(* CODESYS project Brau-Codesys
   Author: Robert Budgen
   Company: Burkert-Canada
   CompiledLibraryCompatibilityVersion: e!COCKPIT
   DefaultNamespace: Brau
   LanguageModelAttribute: qualified-access-only
   Placeholder: Brau
   Title: Brau
   Version: 3.0.0.49

Project tree, tasks and I/O mapping:
  libraries: CAA Types Extern, 3.5.17.0 (CAA Technical Workgroup); CAA Behaviour Model, 3.5.19.0 (CAA Technical Workgroup); CAA FB Factory, 3.5.19.0 (CAA Technical Workgroup); Standard, 3.5.18.0 (System); Util, 3.5.21.0 (System); CmpBitmapPool, 3.5.17.0 (System); VisuDialogs, * (System); MemoryUtils, 3.5.18.0 (3S - Smart Software Solutions GmbH); CAA Memory, 3.5.17.0 (CAA Technical Workgroup); SysTimeRtc, 3.5.20.0 (System); CAA CiA 405, 4.1.0.0 (CAA Technical Workgroup); IoDrvEtherNetIPAdapter, 4.8.0.0 (CODESYS); IoDrvEtherNetIP, 4.8.0.0 (CODESYS); BUILDING, 1.0.0.0 (OSCAT); BASIC, 3.3.4.0 (OSCAT); FloatingPointUtils, 4.0.0.0 (System); 3S CANopenStack, 4.3.0.0 (CODESYS); IoDrvModbusTCP, 4.5.0.0 (CODESYS); Recipe Management, * (System); Burkert Device Library, 1.0.0.102 (Burkert)
  25 Interfaces/
    interface IcSensorProvider: GetSensorRef
  50 Functions/
    Burkert Library/
      function Alarm_Window_Convert [ST]
      function ASi_8694_Mapping [CFC]
      function block b8619_CND_FB [ST]
      function block B8619_Input_FB [ST]
      function block B8619_Main_FB [ST]
      function block b8619_PH_ORP_FB [ST]
      function Build_ORF_Index [ST]
      function FlowWave_Mapping [LD]
      function Tempered_Look_UP [ST]
    function DaySeconds [?]
  90 Task Enums/
    data type eCLT_Task
    data type eGR_Task
    data type eHLT_Task
    data type eKT_Task
    data type eLT_Task
    data type eMM_Task
    data type eWP_Task
    Level_3/
  95 Base Mappings/
    Level_0/
      data type IoLink_Mapping
      data type ME44AI_Mapping
      data type ME44AO_Mapping
      data type ME44DI_Mapping
      data type ME44DO_Mapping
      data type me64_Mapping
    Level_1/
      data type ACV_Mapping_1
      data type AIT_Mapping_1
      data type b8653_mapping
      data type BCV_Mapping_1
      data type cSensor_Mapping
      data type dACV_Mapping
      data type dBCV_Mapping
      data type DI_Mapping
      data type Do_Mapping
      data type FIT_Mapping_1
      data type LS_Mapping_1
      data type PT_Mapping_1
      data type s8050_Mapping
      data type s8228_Mapping
      data type s8312_Mapping
      data type s8412_Mapping
      data type SV_Mapping
      data type TT_Mapping_1
      data type v336x_Mapping
    Level_2/
      data type Analog_Pump_Mapping
      data type mPump_Mapping
      data type PID_Mapping_1
      data type Stack_Light_Mapping
      data type VFD_Mapping
    Level_3/
      data type Alarm_Offset_Mapping
      data type Brite_Mapping_1
      data type Fermenter_Mapping_1
  AL1342
  CanOpen_8694
  Level_3/
    Fermenter
  function block ACV_Temp_Loop_UDFB [CFC]
  function block AODD_UDFB [CFC]
  Asi/
    function block AC2916_AIT [LD]
    function block ACV_ASI_CTRL_UDFB [?]
    function block B8681_ASI_UDFB [CFC]
    function block BCV_ASI_CTRL_UDFB [?]
  function block Basic_Temp_LOOP [CFC]
  function block BCV_Temp_Loop_UDFB [CFC]
  Burkert Library/
    Burkert/
      function eDip_ME44_AO [ST]
      function eDip_ME44_DO_Analog [ST]
      function eDip_ME44_DO [ST]
      function block eDip_ReadSingleItem [ST]
      function block ME43_SDO [ST]: Direct_Write
      function ME44_DI [ST]
    CanOpen/
    eDip/
      function block eDip_8605_CTRL [ST]: Parse_TX
      function eDip_ME44_AI [ST]
      function eDip_ME44_DI [ST]
    function block Parse_DDO [ST]
    function block Parse_DSO [ST]
  function block Chase_Master_Rate_UDFB [SFC]
  function block Chase_Master_UDFB [SFC]
  function block Chase_Slave_UDFB [ST]
  Level_0_Remote_IO/
    function block AL1340_UDFB [ST]
    function block AL1342_UDFB [ST]
    MicroControl/
      function MC4AI [ST]
  Level_1_Devices/
    function block Analog_Control_UDFB [LD]
    Burkert Library/
      function block Analog_Alarm_UDFB [ST]: run
      function block Analog_Sensor_UDFB [?]
      function block B8619_UDFB [CFC]: PH
      function block Basic_ACV_UDFB [?]
      function block Basic_BCV_UDFB [ST]: Eval_Output, Eval_Ready, Eval_Status
      function block Basic_FIT [?]
      function block BCV_CTRL_UDFB [?]
      CanOpen/
        function block CanOpen_8098 [CFC]
        function block CanOpen_8228 [ST]
        function block CanOpen_8691 [?]
        function block CanOpen_8694 [?]
        function block CanOpen_MS02 [ST]
        function block CanOpen_MS03 [ST]
        function block CanOpen_MS04 [ST]
        function block CanOpen_MS05 [ST]
      eDip/
        function block eDip_336x [ST]
        function block eDip_8098_CTRL [ST]
        function block eDip_8228_MEx3 [ST]
        function block eDip_8312 [ST]
        function block eDip_8412 [ST]
        function block eDip_8681_UDFB [CFC]
        function block eDIP_SDO_Manager [CFC]
      function block FIT_Count_UDFB [?]
      function block FIT_Rate_UDFB [?]
      function block FIT_UDFB [?]
      IoLink/
        function block s8050_UDFB [CFC]
      function block LS_UDFB [ST]
      function SV_Fun [CFC]
    function block Stack_Lights_4Way [CFC]
  Level_2_Controls/
    function block Analog_Batch_Pump [CFC]: Set_Status
    function block Batch [ST]: AUX
    function block Condensate_Trap_UDFB [CFC]: Positions, Purge, Status
    function block DofMaster [ST]
    function block Duplex_VFD [ST]: Outputs
    function block PID_UDFB [CFC]
    function block Quick_Mix_UDFB [SFC]: Auto_active, Aux_active, End_active, FIT_Reset_active, Init_active, Init_entry, Main_Rate_active, OFF_active, OFF_entry, Paused_active, Ramp_Down_active, Ramp_Up_active, Start_active, Start_entry, System_Test_active, System_Text_entry
    function block Rate_Batch [ST]
    function block SW_CTRL_ACV [ST]
    function block SW_CTRL [ST]
    function block Tempered_Line_4_Valve [ST]: Alarms, AUX, Math, PID_CTRL, Task_Calibrate, Task_Prime, Task_Run
  Level_3/
  program PLC_TIME [ST]
  Simulators/
    function block c8691_CanOpen_Sim [ST]
    function c8694_CanOpen_Sim [ST]
    function CanOpen_8694_Data_Sim [ST]
    function block Contactor_Sim [ST]
    function Edip_8691_Sim [ST]
    function Edip_8694_Data_Sim [ST]
    function eDip_ME44_DI_Count_Sim [ST]
    function eDip_ME44_DI_Hz_Sim [ST]
    function FIT_Sim [ST]
    function Mix_Sim [ST]
    function TT_SIM [ST]
    function block Vacon_VFD_SIM [ST]
  function block Tempered_Mix_eDip_UDFB [CFC]
  function block Tempered_Mix_UDFB [CFC]
  function block Transfer_ACV_FIT_UDFB [CFC]
  function block Transfer_ACV_VFD_FIT_UDFB [CFC]
  function block Transfer_BCV_FIT_UDFB [CFC]
  function block Transfer_BCV_VFD_FIT_UDFB [CFC]
  Vessels/
  In Burkert Device Library/
    Base_Declarations/
      data type cBase_FIT
      Level_1/
    Level_0_Remote_IO/
    LeveL_1/
      data type cACV
      data type cAIT
      data type cAnalog_Sensor
      data type cBCV
      data type cFIT
      IO-Link/
        data type c8050
      Networked/
      data type SV_DUT
    To be Sorted/
      data type ACV_eDip
      data type Alarm_Config
      data type Alarm_Window
      data type Analog_scale
      data type AODD_DUT
      data type Asi_Node_DUT
      data type b8619_CND_DUT
      data type b8619_Inputs_DUT
      data type b8619_Main_DUT
      data type b8619_PH_DUT
      data type B8691_Asi_DUT
      data type c8694_PDin
      data type cFLOWave_DUT
      data type CND_8619
      data type cSDO_DUT
      data type eDip_8681_DUT
      data type eDip_DDO
      data type eDip_DSO
      data type eDip_MFC_DUT
      data type FV_DUT
      data type HLT_Blending_DUT
      data type HLT_Chase_DUT
      data type PH_8619
      data type PT_Config_DUT
      data type SDO
      data type Steam_Set_Config_DUT
      data type Steam_Set_DUT
      data type TT_Config_DUT
      data type Vessel_Config_Dut
      data type Word_as_Real_DUT
  Level_0/
    Adam_6050/
      data type cAdam_6050_MBTCP
    Adam_6052/
      data type cAdam_6052_Control
      data type cAdam_6052_MBTCP
    Adam_6217/
    Adam_6250/
    IO-Link/
      data type c8694_Io_Link
      data type cIFM_AL1340
      data type cIFM_AL1342
    data type MicroControl_4AI
    SIO-MB04RTDS/
      data type cMB0_RTD
    SIO-MB12CDR/
      data type cSIO_MB12CDR
  Level_1_Devices/
    data type cContactor
    data type DI_DUT
  Level_2_Functions/
    data type Analog_Control_DUT
    data type cAnalog_Batch_Pump
    data type cCondensate_Trap
    data type cDuplex
    data type cFilters
    data type cStack_Light
  Level_3/
    Brewery/
      data type Brewery_Config_DUT
    data type cBatch
    data type cDOF_Master
  Burkert Library/
    data type IFM_Status
    data type ORF
    data type uACV_Mode
    data type uACV_Status
    data type uAIT_Mode
    data type uBCV_Mode
    data type uNamur
    data type uNord_Data_In
    data type uNord_Status_Word
    data type uSensor_Status
  data type Bytes_2_Int
  data type bytes_2_real
  data type Bytes_DWord
  data type Bytes_Word
  data type eKT_Mode
  Level_1/
    data type uAnalog_Pump_Modes
    data type uAnalog_Pump_Status
    data type uContactor_Modes
    data type uDI_Mode
    data type uDI_Status
    data type uDo_Modes
    data type uHOA_Mode
    data type uM_Pump_Modes
    data type uM_Pump_Status
    data type uVFD_Mode
    data type uVFD_Status
  data type REAL_2_WORD
  data type uBatch_Status
  data type uBatch_Task
  data type uBatch_Transfer_Mode
  data type uBrite_Modes
  data type uBrite_Status
  data type uBrite_Status
  data type uChase_Status
  data type uCLT_Mode
  data type uCLT_Status
  data type uCLT_Task
  data type uContactor_Status
  data type uFermenter_Modes
  data type uFermenter_Status
  data type uFilter_Manager_Modes
  data type uFilterMode
  data type uGR_Status
  data type uGR_Task
  data type uHighSpeed_Tempered_Mode
  data type uHighSpeed_Tempered_Status
  data type uHighSpeed_Tempered_Task
  data type uHLT_Mode
  data type uHLT_Status
  data type uHLT_Task
  data type uKT_Mode
  data type uKT_Status
  data type uKT_Task
  data type uLT_Mode
  data type uLT_Status
  data type uLT_Task
  data type uMM_Mode
  data type uMM_Task
  data type uPID_Modes
  data type uPID_Status
  data type uQuick_Mix_Modes
  data type uService_Water_Destination
  data type uTempered_Modes
  data type uTempered_Status
  data type uTempered_Tasks
  data type uUser_Confirm
  data type uWP_Mode
  data type uWP_Modes
  data type uWP_Status
  data type uWP_Task
  data type WORD_2_Real
  data type AIT_Transfer_Modes
  Burkert Library/
    Brewery/
    data type e_8681_Modes
    data type eAODD_Modes
    data type eB336x_Modes
    data type eConfig_startTune
    data type eHOA_Modes
    Level_1/
      data type ACV_Modes
      data type AIT_Modes
      data type eBCV_Modes
      data type TT_Modes
    data type LS_Modes
    data type Positioner_Modes
    data type PT_Modes
    data type Reset_Relay_Mode
  data type CLT_Modes
  data type Command_Modes
  data type eChase_Mode
  data type Fan_Modes
  data type FIT_Transfer_Modes
  data type FIT_VFD_Transfer_Modes
  Level_0/
  Level_1/
    data type eVFD_Modes
  Level_3/
    data type eBrite_Modes
    data type eCLT_Modes
    data type eFermenter_Modes
    data type eGR_Modes
    data type eHLT_Modes
    data type eKT_Modes
    data type eLT_Modes
    data type eMM_Modes
    data type eRCP_Mode
    data type eWP_Modes
    data type FV_Modes
    data type HLT_Blending_Modes
    data type KTWP_Modes
  data type Steam_Condensate_Modes
  data type Steam_Modes
  data type Temp_loop_Modes
  Burkert Library/
    Level_1/
      data type eACV_Status
      data type eBCV_Status
      data type eSensor_Status
  data type e8691_ValveMode
  data type e8691_xTuneStatus
  data type e8694_xTuneStatus
  data type eB8681_Status
  data type eCurrentOpMode
  data type eNamur107
  data type eORF_Status
  Level_1/
    data type Contactor_Status
    data type DI_Status
    data type DO_Status
    data type eAnalog_Pump_Status
    data type eAODD_Status
    data type eM_Pump_Status
    data type eVFD_Status
    data type VFD_Fault_Status
  Level_2/
    data type eCondensate_Status
    data type eFilter_Manager_Status
    data type eFilter_Status
  Level_3/
  data type SDO_Error_Codes
  Vessels/
    data type eBrite_Status
    data type eCLT_Status
    data type eHLT_Status
    data type eKT_Status
    data type eLT_Status
    data type eMM_Status
    data type eWP_Status
  data type eHLT_Notifications
  data type eMM_Notifications
  function GetLibVersion [ST]
  function GetLibVersionNumber [ST]
  function IsLibReleased [ST]
  function GetBooleanProperty [ST]
  function GetCompany [ST]
  function GetTextProperty2 [ST]
  function GetTextProperty [ST]
  function GetTitle [ST]
  function GetVersion [ST]
  function GetVersionProperty [ST]
  function block FB_PositionTracker [ST]
  function fbMidPoint [ST]
  function RCP_Manager [ST]
  function block Virtual_FIT [CFC]
  Burkert Library/
    ASi/
      function block ASi_8694_HMI_Sync_UDFB [?]
    Level_0/
    Level_1/
      function block ACV_HMI_Sync_UDFB [?]
      function block AIT_HMI_Sync_UDFB [?]
      function block B8050_HMI_Sync_UDFB [?]
      function block BCV_HMI_Sync_UDFB [?]
      function block c8691_HMI_Sync_UDFB [?]
      function block c8694_HMI_Sync_UDFB [?]
      function block DI_HMI_Sync_UDFB [?]
      function block FIT_HMI_Sync_UDFB [?]
      function block GS20_VFD_HMI_Sync [?]
      function block s336x_HMI_Sync [?]
      function block s8050_HMI_Sync [?]
      function block s8098_HMI_Sync_UDFB [?]
      function block s8312_HMI_Sync [?]
      function block SV_HMI_Sync [?]
      function block Vacon_HMI_Sync_UDFB [?]
  Level_1/
    function block Analog_Pump_HMI_Sync [?]
    function block Contactor_HMI_Sync_UDFB [?]
    function block Eaton_VFD_HMI_Sync [?]
    function block M_Pump_HMI_Sync [?]
  Level_2/
    function block PID_HMI_Sync_UDFB [?]
  Level_3/
    function block Brite_HMI_Sync [?]
    function block Fermenter_HMI_Sync [?]
  data type ASi_8694
  data type ASi_8694_PDO
  Burkert Librarry/
    Level_0/
    Level_1/
      data type HMI_8050
      data type HMI_AIT
      data type HMI_BCV
      data type HMI_FIT
      data type HMI_VFD_GS20_DUT
      data type HMI_VFD_Vacon_DUT
  Level_1/
    data type HMI_Analog_Pump
    data type HMI_Contactor_DUT
    data type HMI_M_Pump
    data type HMI_VFD_Eaton_DUT
  Level_2/
    data type HMI_PID
  Level_3/
    data type HMI_Brite
    data type HMI_Fermenter
  function block AC2916 [CFC]
  function block Asi_GW_FUN [ST]
  function f_Fermenter_To_NVL [ST]
  data type eAnalog_Control_Modes
  data type eFilter_Manager_Modes
  data type eFilter_Mode
  data type eTempered_Modes
  function Adam_6050_FB [LD]
  function Adam_6250 [ST]
  function block MB0_RTD [ST]
  function block SIO_MB12CDR [ST]
  function block Contactor [ST]: Status
  function block Contactor_Control_UDFB [CFC]: Status
  function block DI_UDFB [CFC]
  function block DO_UDFB [CFC]
  function block Analog_Pump [ST]: Status
  function block Eaton_DM1 [ST]: Control, Data_IN, Data_Out, Status
  function block Nord_VFD_UDFB [CFC]
  function block Vacon_100 [ST]: Control, Data_IN, Data_Out, Data_Sim, Status
  function block VFD_GS20_UDFB [?]: Status
  function block VFD_GS2_UDFB [LD]
  function block VFD_Vacon100_UDFB [?]
  function block Wago_750_455 [LD]
  function block Wago_750_NAMUR_NE43 [?]
  data type VFD_CONTROL
  data type VFD_GS2_DUT
  data type VFD_WEG_DUT
  data type cFilter
  data type cFilter_Manager
  data type Quick_Mix_Control
  data type cPID_DUT
  data type cTempered_Line_Data
  function block Brite_1_UDFB [CFC]
  function block Brite_2_UDFB [CFC]
  function block Brite_3_UDFB [CFC]
  function block Fermenter_1_UDFB [CFC]
  function block Fermenter_2_UDFB [CFC]
  function block Fermenter_3_UDFB [CFC]
  program CLT [ST]
  KT/
  LT/
  MM/
  WP/
  program Grain_Room_Hopper_1Conveyor [ST]
  Controls/
  program HLT_2Pump_2Mix [ST]
  program HLT_2Pump_2Mix_OLD [CFC]
  function block HLT_PID_Manager [CFC]
  function block HLT_Status_Manager [?]
  function block HLT_Task_Manager [CFC]
  function block HLT_Tasks_OLD [SFC]
  function block HLT_Valve_Manager [CFC]
  function block HLT_VFD_Ctrl [CFC]
  function block Service_Water [SFC]
  function block Service_Water_Manager [CFC]
  Tasks/
  data type ceDip_ME44_DI
  data type cME44_DO
  data type cME44_DO_TX
  data type cVFD_Eaton_DUT
  data type cNord_VFD
  data type cVFD_STATUS_Vacon
  data type cVFD_Vacon
  data type cCellar_Vessel_Config_DUT
  program CIP_CTRL [LD]
  program CIP_PID_CTRL [CFC]
  program CIP_Pump_CTRL [CFC]
  program CIP_Valve_CTRL [CFC]
  data type cVessel_CIP
  data type cCLT_Assets
  data type CLT_DUT
  data type CLT_Profile
  data type eCLT_Profile
  data type Heat_Profile_DUT
  data type GR_DUT
  data type Grain_Room_Assets
  data type eHLT_Profile
  data type eHLT_Setpoints
  data type HLT_Assets
*)

// Bytes_2_Int
TYPE Bytes_2_Int :
UNION
	Raw:ARRAY[0..1] OF BYTE;
	qInt:INT;
END_UNION
END_TYPE

// bytes_2_real
TYPE bytes_2_real :
UNION
	Raw_bytes:ARRAY[0..3] OF BYTE;
	value:REAL;
END_UNION
END_TYPE

// Bytes_DWord
TYPE Bytes_DWord :
UNION
	tByte:ARRAY[0..3] OF BYTE;
	tUSINT:ARRAY[0..3] OF USINT; 
	tInt:ARRAY[0..1] OF INT;
	tuInt:ARRAY[0..1] OF UINT;
	tWord:ARRAY[0..1] OF WORD;
	tReal:REAL;
	tDint:DINT;
	tUDINT:UDINT;
	tDword:DWORD;
	//tString:STRING(4);
	
END_UNION
END_TYPE

// Bytes_Word
TYPE Bytes_Word :
UNION
	tByte:ARRAY[0..1] OF BYTE;
	tWord: WORD;
	tInt:INT;
	tUint:UINT;
END_UNION
END_TYPE

// eKT_Mode
TYPE eKT_Mode :
UNION
	iMode:INT;
	eMode:eKT_Modes;
END_UNION
END_TYPE

// REAL_2_WORD
TYPE REAL_2_WORD :
UNION
	rReal:REAL;
	wWord:ARRAY[0..1]OF WORD;
END_UNION
END_TYPE

// uBatch_Status
TYPE uBatch_Status :
UNION
	iStatus:INT;
	eStatus:eBatch_Status;
END_UNION
END_TYPE

// uBatch_Task
TYPE uBatch_Task :
UNION
	iTask:INT;
	eTask:eBatch_Task;
END_UNION
END_TYPE

// uBatch_Transfer_Mode
TYPE uBatch_Transfer_Mode :
UNION
	iMode:INT;
	eMode:eBatch_Transfer_Mode;
END_UNION
END_TYPE

// uBrite_Modes
TYPE uBrite_Modes :
UNION
	iMode:INT;
	eMode:eBrite_Modes;
END_UNION
END_TYPE

// uBrite_Status
TYPE uBrite_Status :
UNION
	eStatus:eBrite_Status;
	iStatus:INT;
END_UNION
END_TYPE

// uBrite_Status
TYPE uBrite_Status :
UNION
	eStatus:eBrite_Status;
	iStatus:INT;
END_UNION
END_TYPE

// uChase_Status
TYPE uChase_Status :
UNION
	iStatus:INT;
	eStatus:eChase_Status;
END_UNION
END_TYPE

// uCLT_Mode
TYPE uCLT_Mode :
UNION
	iMode:INT;
	eMode:eCLT_Modes;
END_UNION
END_TYPE

// uCLT_Status
TYPE uCLT_Status :
UNION
	iStatuus:INT;
	eStatus:eCLT_Status;
END_UNION
END_TYPE

// uCLT_Task
TYPE uCLT_Task :
UNION
	iTask:INT;
	eTask:eCLT_Task;
END_UNION
END_TYPE

// uContactor_Status
TYPE uContactor_Status :
UNION
	eStatus:eContactor_Status;
	iStatus:INT;
END_UNION
END_TYPE

// uFermenter_Modes
TYPE uFermenter_Modes :
UNION
	iMode:INT;
	eMode:eFermenter_Modes;
END_UNION
END_TYPE

// uFermenter_Status
TYPE uFermenter_Status :
UNION
	eStatus:eFermenter_Status;
	iStatus:INT;
END_UNION
END_TYPE

// uFilter_Manager_Modes
TYPE uFilter_Manager_Modes :
UNION
	iMode:INT;
	eMode:eFilter_Manager_Modes;
END_UNION
END_TYPE

// uFilterMode
TYPE uFilterMode :
UNION
	iMode:INT;
	eMode:eFilter_Mode;
END_UNION
END_TYPE

// uGR_Status
TYPE uGR_Status :
UNION
	iStatuus:INT;
	eStatus:eGrain_Room_Status;
END_UNION
END_TYPE

// uGR_Task
TYPE uGR_Task :
UNION
	iTask:INT;
	eTask:eGR_Task;
END_UNION
END_TYPE

// uHighSpeed_Tempered_Mode
TYPE uHighSpeed_Tempered_Mode :
UNION
	iMode:INT;
	eMode:eHighSpeed_Tempered_Mode;
END_UNION
END_TYPE

// uHighSpeed_Tempered_Status
TYPE uHighSpeed_Tempered_Status :
UNION
	iStatus:INT;
	eStatus:eHighSpeed_Tempered_Status;
END_UNION
END_TYPE

// uHighSpeed_Tempered_Task
TYPE uHighSpeed_Tempered_Task :
UNION
	iTask:INT;
	eTask:eHighSpeed_Tempered_Task;
END_UNION
END_TYPE

// uHLT_Mode
TYPE uHLT_Mode :
UNION
	iMode:INT;
	eMode:eHLT_Modes;
END_UNION
END_TYPE

// uHLT_Status
TYPE uHLT_Status :
UNION
	iStatuus:INT;
	eStatus:eHLT_Status;
END_UNION
END_TYPE

// uHLT_Task
TYPE uHLT_Task :
UNION
	iTask:INT;
	eTask:eHLT_Task;
END_UNION
END_TYPE

// uKT_Mode
TYPE uKT_Mode :
UNION
	iMode:INT;
	eMode:eKT_Modes;
END_UNION
END_TYPE

// uKT_Status
TYPE uKT_Status :
UNION
	iStatuus:INT;
	eStatus:eKT_Status;
END_UNION
END_TYPE

// uKT_Task
TYPE uKT_Task :
UNION
iTask:INT;
eTask:eKT_Task;
END_UNION
END_TYPE

// uLT_Mode
TYPE uLT_Mode :
UNION
	iMode:INT;
	eMode:eLT_Modes;
END_UNION
END_TYPE

// uLT_Status
TYPE uLT_Status :
UNION
	eStatus:eLT_Status;
	iStatus:INT;
END_UNION
END_TYPE

// uLT_Task
TYPE uLT_Task :
UNION
iTask:INT;
eTask:eLT_Task;
END_UNION
END_TYPE

// uMM_Mode
TYPE uMM_Mode :
UNION
	iMode:INT;
	eMode:eMM_Modes;
END_UNION
END_TYPE

// uMM_Task
TYPE uMM_Task :
UNION
	iTask:INT;
	eTask:eMM_Task;
END_UNION
END_TYPE

// uPID_Modes
TYPE uPID_Modes :
UNION
	iMode:INT;
	eMode:ePID_Modes;
	
END_UNION
END_TYPE

// uPID_Status
TYPE uPID_Status :
UNION
	iStatus:INT;
	eStatus:ePID_Status;
END_UNION
END_TYPE

// uQuick_Mix_Modes
TYPE uQuick_Mix_Modes :
UNION
	iMode:INT;
	eMode:eQuick_Mix_Modes;
END_UNION
END_TYPE

// uService_Water_Destination
TYPE uService_Water_Destination :
UNION
	iTarget:INT;
	eTarget:Service_Water_Mapping;
END_UNION
END_TYPE

// uTempered_Modes
TYPE uTempered_Modes :
UNION
	iMode:INT;
	eMode:eTempered_Modes;
END_UNION
END_TYPE

// uTempered_Status
TYPE uTempered_Status :
UNION
	iStatus:INT;
	eStatus:eTempered_Status;
END_UNION
END_TYPE

// uTempered_Tasks
TYPE uTempered_Tasks :
UNION
	iTask:INT;
	eTask:eTempered_Task;
END_UNION
END_TYPE

// uUser_Confirm
TYPE uUser_Confirm :
UNION
	iConfirm:INT;
	eConfirm:eUser_Confirm;
	
END_UNION
END_TYPE

// uWP_Mode
TYPE uWP_Mode :
UNION
	iMode:INT;
	eMode:eWP_Modes;
END_UNION
END_TYPE

// uWP_Modes
TYPE uWP_Modes :
UNION
	iMode:INT;
	eMode:eWP_Modes;
END_UNION
END_TYPE

// uWP_Status
TYPE uWP_Status :
UNION
	iStatus:INT;
	eStatus:eWP_Status;
END_UNION
END_TYPE

// uWP_Task
TYPE uWP_Task :
UNION
	iTask:INT;
	eTask:eWP_Task;
END_UNION
END_TYPE

// WORD_2_Real
TYPE WORD_2_Real :
UNION
	wWord:ARRAY[0..1] OF WORD;
	rReal:REAL;
	
END_UNION
END_TYPE

// AIT_Transfer_Modes
{attribute 'qualified_only'}
//{attribute 'strict'}
TYPE AIT_Transfer_Modes :
(
	Idle := 0,
	Maintain_Target,
	//Flow_Only,
	Hz_only,
	//Pressure_Only,
	//LS_Dry,
	//Flow_Timed,
	Timed,
	Hz_Timed,
	//Pressure_Timed,
	//Batch,
	Lock_Out,
	Passive,
	Pause,
	Resume
	);
END_TYPE

// CLT_Modes
{attribute 'qualified_only'}
//{attribute 'strict'}
TYPE CLT_Modes :
(
	Off := 0,
	Auto_Run,
	Auto_Paused,
	Auto_Halt
	
);
END_TYPE

// Command_Modes
{attribute 'qualified_only'}
//{attribute 'strict'}
TYPE Command_Modes :
(
	Off := 0,
	Auto_Run,
	Auto_Paused,
	Auto_Complete,
	Auto_Halt
	
);
END_TYPE

// eChase_Mode
{attribute 'qualified_only'}
//{attribute 'strict'}
{attribute 'to_string'}
TYPE eChase_Mode :
(
	Auto := 0,
	OFF,
	Manual
);
END_TYPE

// Fan_Modes
{attribute 'qualified_only'}
//{attribute 'strict'}
TYPE Fan_Modes :
(
	Off := 0,
	On,
	Auto
	
);
END_TYPE

// FIT_Transfer_Modes
{attribute 'qualified_only'}
//{attribute 'strict'}
TYPE FIT_Transfer_Modes :
(
	Idle := 0,
	//AIT_Only,
	//Flow,
	//Hz_only,
	//Pressure_Only,
	//LS_Dry,
	//Flow_Timed,
	//AIT_Timed,
	//Hz_Timed,
	//Pressure_Timed,
	Batch,
	Lock_Out,
	Passive,
	Pause,
	Resume
	);
END_TYPE

// FIT_VFD_Transfer_Modes
{attribute 'qualified_only'}
//{attribute 'strict'}
TYPE FIT_VFD_Transfer_Modes :
(
	Idle := 0,
	//AIT_Only,
	//Flow_Only,
	//Hz_only,
	//Pressure_Only,
	//LS_Dry,
	//Flow_Timed,
	//AIT_Timed,
	//Hz_Timed,
	//Pressure_Timed,
	Batch,
	Lock_Out,
	Passive,
	Pause,
	Resume
	);
END_TYPE

// Steam_Condensate_Modes
{attribute 'qualified_only'}
//{attribute 'strict'}
TYPE Steam_Condensate_Modes :
(
	Ready := 0,
	Condensdate_Return
	
);
END_TYPE

// Steam_Modes
{attribute 'qualified_only'}
//{attribute 'strict'}
TYPE Steam_Modes :
(
	Off := 0,
	Blow_Down,
	Ready
	
);
END_TYPE

// Temp_loop_Modes
{attribute 'qualified_only'}
//{attribute 'strict'}
TYPE Temp_loop_Modes :
(
	Idle := 0,
	Crash,
	Profile,
	Step,
	Auto,
	Auto_Paused
);
END_TYPE

// e8691_ValveMode
{attribute 'qualified_only'}
//{attribute 'strict'}
{attribute 'to_string'}
TYPE e8691_ValveMode :
(

	Init:=0,
	Normal,
	Tune,
	Safe
	
);
END_TYPE

// e8691_xTuneStatus
{attribute 'qualified_only'}
//{attribute 'strict'}
{attribute 'to_string'}
TYPE e8691_xTuneStatus :
(
	Ready:=0,
	Init,
	POS1,
	POS2,
	Stroke,
	SwTimes,
	
	errAbort:=250,
	errSafePos:=251,
	errSwTimes:=252,
	errStroke:=253,
	errPos2:=254,
	errPos1:=255
);	
END_TYPE

// e8694_xTuneStatus
{attribute 'qualified_only'}
//{attribute 'strict'}
{attribute 'to_string'}
TYPE e8694_xTuneStatus :
(
	Complete := 0,
	Ready,
	Init,
	EndStops,
	Leakage,
	Offset,
	Friction,
	Controller,
	NeverRan:=127,
	errTurnPoti:=250,
	errLeakageYB:=251,
	errLeakage:=252,
	errTimeOut:=253,
	errBreakErr:=254,
	errBreakUser:=255
);	
END_TYPE

// eB8681_Status
{attribute 'qualified_only'}
//{attribute 'strict'}
TYPE eB8681_Status :
(	
	Unknown:=0,
	Blocked,
	Open,
	Upper_Drain,
	Lower_Drain,
	Missing,
	Detected,
	P_Fault
);
END_TYPE

// eCurrentOpMode
{attribute 'qualified_only'}
//{attribute 'strict'}
{attribute 'to_string'}
TYPE eCurrentOpMode :
(
	xControl := 1,
	CutOffUp,
	CutOffDn,
	SafePosUp,
	SafePosDn,
	SafePos,
	Manual,
	xTune
	
);
END_TYPE

// eNamur107
{attribute 'qualified_only'}
//{attribute 'strict'}
{attribute 'to_string'}
TYPE eNamur107 :
(
	Normal := 0,			//White
	OK,						//Green
	MaintenanceReq,			//Blue
	OutOfSpec,				//Yellow
	Warning,				//Orange
	Error,					//Red
	
	Offline:=10				//black
	
);
END_TYPE

// eORF_Status
{attribute 'qualified_only'}
//{attribute 'strict'}
TYPE eORF_Status :
(
	NoError:=16#00,
	GeneralError:=16#02,
	No_Subindex_specifed:=16#04,
	Access_NOT_supported:=16#05,
	Data_length_too_great:=16#09,
	Data_length_too_small:=16#0A,
	No_object:=16#0F,
	Service_could_not_be_implemented:=16#11,
	Read_access_only:=16#1F,
	No_data:=16#21,
	No_device_with_this_Node_ID_available:=16#FF,
	Processisrunning:=16#FFFF
);
END_TYPE

// SDO_Error_Codes
{attribute 'qualified_only'}
{attribute 'strict'}
TYPE SDO_Error_Codes :
	(
	Dummy:=0
(*
	 SDO_ERR_TOGGLE_BIT   :=16#05030000,
 
 	SDO_ERR_TIMEOUT   :=16#05040000,
 
 	SDO_ERR_COMMAND   :=16#05040001,
 
 	SDO_ERR_BLOCK_SIZE   :=16#05040002,
 
 	SDO_ERR_BLOCK_SEQUENCE   :=16#05040003,
 
 	SDO_ERR_BLOCK_CRC   :=16#05040004,
 
 	SDO_ERR_MEMORY   :=16#05040005,
 
 	SDO_ERR_ACCESS_UNSUPPORTED   :=16#06010000,
 
 	SDO_ERR_ACCESS_WO   :=16#06010001,
 
 	SDO_ERR_ACCESS_RO   :=16#06010002
 
 	SDO_ERR_NO_OBJECT   :=16#06020000
 
 	SDO_ERR_MAPPING_OBJECT   :=16#06040041
 
 	SDO_ERR_MAPPING_LENGTH   :=16#06040042
 
 	SDO_ERR_GENERAL_PARAMETER   :=16#06040043
 
 	SDO_ERR_GENERAL_DEVICE   :=16#06040047
 
 	SDO_ERR_HARDWARE   :=16#06060000
 
 	SDO_ERR_DATATYPE   :=16#06070010
 
 	SDO_ERR_DATATYPE_HIGH   :=16#06070012
 
 	SDO_ERR_DATATYPE_LOW   :=16#06070013
 
 	SDO_ERR_NO_SUB_INDEX   :=16#06090011
 
 	SDO_ERR_VALUE_RANGE   :=16#06090030
 
 	SDO_ERR_VALUE_HIGH   :=16#06090031
 
 	SDO_ERR_VALUE_LOW   :=16#06090032
 
 	SDO_ERR_VALUE_MIN_MAX   :=16#06090036
 
 	SDO_ERR_SDO_CONNECTION   :=16#060A0023
 
 	SDO_ERR_GENERAL   :=16#08000000
 
 	SDO_ERR_DATA_STORE   :=16#08000020
 
 	SDO_ERR_DATA_STORE_LOCAL   :=16#08000021
 
 	SDO_ERR_DATA_STORE_STATE   :=16#08000022
 
 	SDO_ERR_OBJECT_DICTIONARY   :=16#08000023
 
 	SDO_ERR_NO_DATA   :=16#08000024
*)
);
END_TYPE

// 90 Task Enums/eCLT_Task
{attribute 'qualified_only'}
//{attribute 'strict'}
{attribute 'to_string'}
TYPE eCLT_Task :
(
	Off :=0,						
	Fill, 													
	Cool_Recirculate,
	Ready_Holding,		//3
	Ready,		
	Line_Chase,				
		
	Spray_Ball,
	Fill_Cool
		

	
);
END_TYPE

// 90 Task Enums/eGR_Task
{attribute 'qualified_only'}
//{attribute 'strict'}
{attribute 'to_string'}
TYPE eGR_Task :
(
	OFF := 0,
	Dispense
);
END_TYPE

// 90 Task Enums/eHLT_Task
{attribute 'qualified_only'}
//{attribute 'strict'}
{attribute 'to_string'}
TYPE eHLT_Task :
(
	Off :=0,						
	Fill, 													
	Heat_Recirculate,
	Ready_Holding,
	Ready,		
	Line_Chase,				
		
	Spray_Ball,
	Fill_Heat			

	
);
END_TYPE

// 90 Task Enums/eKT_Task
{attribute 'qualified_only'}
//{attribute 'strict'}
{attribute 'to_string'}
TYPE eKT_Task :
(
	OFF := 0,
	Recipe_Copy,
	PreHeat,
	Wort_In,
	Full_Boil,
	Jacket_Boil,
	Rocket_Boil,
	Transfer,
	Transfer_Chase,
	Quick_Rinse, //8
	Tank_Drain,
	Transfer_in,
	Whirlpool,
	Rest,
	Transfer_Out,
	Turb_Buster, //14
	Drain,		//15
	Mash_In_Rocket_Transition,
	Mash_In_Rocket
);
END_TYPE

// 90 Task Enums/eLT_Task
{attribute 'qualified_only'}
//{attribute 'strict'}
{attribute 'to_string'}
TYPE eLT_Task :
(
	Off :=0,
	Move_Brew_Configuration,	//
	Foundation_Water,
	Mash_In,
	
	First_Underlet,	//4
	Second_Underlet,
	Third_Underlet,
	
	First_Vorlauf,	//7
	Second_Vorlauf,
	Third_Vorlauf,
	
	First_Transfer,	//10
	Second_Transfer,
	Third_Transfer,
	
	First_Sparge,	//13
	Second_Sparge,
	Third_Sparge,
	
	Transfer_Empty,	//16
	Transfer_Chase,		//17
	Tank_Clean,
	Quick_Rinse,		//19
	Tank_Drain,			//20
	Spent_Grain,		//21
	CIP,
	Pre_Heat			//23
	
					
	
	
);
END_TYPE

// 90 Task Enums/eMM_Task
{attribute 'qualified_only'}
//{attribute 'strict'}
{attribute 'to_string'}
TYPE eMM_Task :
(
	Off :=0,					
	Confirm,
	//Confirmed,
	Preheat,
	Mash_In,	//3						
	Heat_1,		//4
	Heat_2,
	Heat_3,
	//Heat_4,
	//Mash_Complete,				
	Mash_Out,		//7			
	//Transfer_Complete,			
	Transfer_Flush,		//8		
	//Transfer_Flush_Complete,	
	Quick_Rinse,	//9			
	//Quick_Rinse_Complete,		
	Drain,			//10			
	//Drain_Complete,				
	
	//CIP_Fill,					
	//CIP_Fill_Complete,			
	//CIP_Recirculate,			
	//CIP_Recirculate_Complete,	
	//CIP_Transfer,				
	//CIP_Transfer_Complete,		
	//CIP_Transfer_Flush,			
	//CIP_Transfer_Flush_Complete 
	CIP,
	Vorlauf,
	Transfer,
	Transfer_Sparge,
	Fly_Sparge,
	UnderLet,
	Foundation,	//17
	Grain_Out,
	CIP_1,
	CIP_2
	

	
	
);
END_TYPE

// 90 Task Enums/eWP_Task
{attribute 'qualified_only'}
{attribute 'to_string'}
TYPE eWP_Task :
(
	Off :=0, 
	Recipe_Copy,					//0
	Transfer_in,
	Whirlpool,
	Rest,
	CastOut,
	CastOut_Chase,
	Trub_Buster,
	Quick_Rinse,
	Tank_Drain
	
);
END_TYPE

// eHLT_Notifications
{attribute 'qualified_only'}
{attribute 'strict'}
TYPE eHLT_Notifications :
(
	System_OK,
	Pump_Not_In_Auto,
	Pump_Faulted,
	HTX_Valve_Not_In_Auto,
	Recirc_Valve_Not_In_Auto,
	Spray_Ball_Valve_Not_In_Auto,
	Refill_Valve_Not_In_Auto,
	Pump_Intake_Empty
	
);
END_TYPE

// eMM_Notifications
{attribute 'qualified_only'}
{attribute 'strict'}
TYPE eMM_Notifications :
(
	System_OK := 0,
	Pump_Fault,
	Pump_Not_In_Auto
);
END_TYPE

// ASi_8694
TYPE ASi_8694 EXTENDS Burkert.cACV :
STRUCT
	PDO:ASi_8694_PDO;
END_STRUCT
END_TYPE

// ASi_8694_PDO
TYPE ASi_8694_PDO :
STRUCT
	Actual:REAL;
	Output:REAL;
END_STRUCT
END_TYPE

// Level_0/MicroControl_4AI
TYPE MicroControl_4AI :
STRUCT
	GW_TCP_State:ModbusTCPComState;
	PV_RX:ARRAY[0..3] OF UINT;
	FV_RX:ARRAY[0..3] OF UINT;
	PV:ARRAY[0..3] OF REAL;
END_STRUCT
END_TYPE

// Level_1_Devices/cContactor
TYPE cContactor :
STRUCT
	Mode:uContactor_Modes;
	Status:uContactor_Status;
	PLC_CMD_FWD:BOOL;
	PLC_CMD_Rev:BOOL;
	Q1:BOOL;
	Q2:BOOL;
	Ready:BOOL;
	
END_STRUCT
END_TYPE

// Level_1_Devices/DI_DUT
TYPE DI_DUT :
STRUCT
	MODE:uDi_Mode;
	Status:uDi_Status;
	Raw:BOOL;
	Q:BOOL;
END_STRUCT
END_TYPE

// Level_2_Functions/Analog_Control_DUT
TYPE Analog_Control_DUT :
STRUCT
	Alarm_Config	:	Burkert.cAlarm_Config;
	Analog_Scale	:	Burkert.cAnalog_scale;
	Mode			:	eAnalog_Control_Modes;
	EU:		REAL;
	PLC_Target:REAL;
	HMI_Target:REAL;
	output:REAL;
	Status:Burkert.eSensor_Status;
END_STRUCT
END_TYPE

// Level_2_Functions/cAnalog_Batch_Pump
TYPE cAnalog_Batch_Pump EXTENDS Burkert.cAnalog_Pump : 
STRUCT
	//Mode:eAnalog_Pump_Modes;
	Config:cAnalog_Batch_Pump_Config;
	HMI_Volume_Target:REAL;
	PLC_Volume_Target:REAL;
	
	Live_Rate:REAL;
	Volume_Delivered:REAL;
	PCT_Remain:REAL;
	Batch_ETA:INT;
	
END_STRUCT
END_TYPE

// Level_2_Functions/cCondensate_Trap
TYPE cCondensate_Trap :
STRUCT
	//LSHH:Burkert.DI_DUT;
	//LSH:Burkert.DI_DUT;
	//LSL:Burkert.DI_DUT;
	//LSLL:Burkert.DI_DUT;
	Min_Valve_Positions:ARRAY[0..3] OF REAL;
	CV:REAL;
	READY:BOOL;
	Status:eCondensate_Status;
END_STRUCT
END_TYPE

// Level_2_Functions/cDuplex
TYPE cDuplex :
STRUCT
	Run_Request:BOOL;
	Run_Pct:REAL;
	Target_Split:REAL;
	Current_Split:REAL;
	
END_STRUCT
END_TYPE

// Level_2_Functions/cFilters
TYPE cFilters :
STRUCT
	Group_Mode:Burkert.uHOA_Mode;
	A_Mode:Burkert.uHOA_Mode;
	A_Status:eFilter_Status;
	A_Task:eFilter_Task;
	
	B_Mode:Burkert.uHOA_Mode;
	B_Status:eFilter_Status;
	B_Task:eFilter_Task;
	
	DP_Alarm:Burkert.cAlarm_Config;
	DP:REAL;
	
	
END_STRUCT
END_TYPE

// Level_2_Functions/cStack_Light
TYPE cStack_Light :
STRUCT
	ON:BOOL;
	Flash_Rate_ms:UINT;
	Q:BOOL;
END_STRUCT
END_TYPE

// Level_3/cBatch
TYPE cBatch :
STRUCT
	Min_Rate:REAL;
	Max_Rate:REAL;
	Start_Volume:REAL;
	End_Volume:REAL;
	
	Batch_Volume:REAL;
	Batch_Rate:REAL;
	
	Live_Target_Volume:REAL;
	Live_Target_Rate:REAL;
	
	Actual_Volume:REAL;
	Actual_Rate:REAL;
	
	
	PCT_Complete:REAL;
	System_Load:REAL;
	ETA:UINT;
	
	Ready:BOOL;
	Active:BOOL;
	
	Line_Mode:Burkert.uHOA_Mode;
	Line_Task:uBatch_Task;
	Line_Status:uBatch_Status;
	PLC_Run:BOOL;
	
	StrLine_Mode:STRING;
	StrLine_Task:STRING;
	StrLine_Status:STRING;
	
	
END_STRUCT
END_TYPE

// Level_3/cDOF_Master
TYPE cDOF_Master :
STRUCT
	
	Batch_Volume:REAL;
	Batch_Rate:REAL;
	Batch_Mode:Burkert.uHOA_Mode;
	Batch_Task:uBatch_Task;
	Batch_Status:uBatch_Status;
	
	PLC_Run:BOOL;
	
	Current_Load_High:REAL;
	Current_Load_Low:REAL;
	Current_Batch_PCT:REAL;
	Batch_CLK:TIME;
	Batch_Remain:TIME;
	Current_Batch_Volume:REAL;
	Current_Batch_Rate:REAL;
	Batch_Target_ms:UDINT;
	Batch_Elapsed_ms:UDINT;
	Batch_Remain_ms:UDINT;
	Batch_ETA_ms:UDINT;
	
	
	StrBatch_Mode:STRING;
	StrBatch_Task:STRING;
	StrBatch_Status:STRING;
	
	MasterID:UDINT:=0;
	Active:BOOL;
	
	
	
	
	
END_STRUCT
END_TYPE

// Burkert Library/IFM_Status
TYPE IFM_Status :
UNION
	RX:WORD;
	Status:ARRAY[0..15] OF BOOL;
END_UNION
END_TYPE

// Burkert Library/ORF
TYPE ORF :
UNION
	Address:DWORD;
	SDO:SDO;
END_UNION
END_TYPE

// Burkert Library/uACV_Mode
TYPE uACV_Mode :
UNION
	iMode:INT;
	eMode:Burkert.eACV_Modes;
END_UNION
END_TYPE

// Burkert Library/uACV_Status
TYPE uACV_Status :
UNION
	iStatus:INT;
	eStatus:eACV_Status;
END_UNION
END_TYPE

// Burkert Library/uAIT_Mode
TYPE uAIT_Mode :
UNION
	iMode:INT;
	eMode:Burkert.AIT_Modes;
END_UNION
END_TYPE

// Burkert Library/uBCV_Mode
TYPE uBCV_Mode :
UNION
	iMode:INT;
	eMode:eBCV_Modes;
END_UNION
END_TYPE

// Burkert Library/uNamur
TYPE uNamur :
UNION
	iNamur:INT;
	eNamur:eNamur107;
	
END_UNION
END_TYPE

// Burkert Library/uNord_Data_In
TYPE uNord_Data_In :
UNION
	
END_UNION
END_TYPE

// Burkert Library/uNord_Status_Word
TYPE uNord_Status_Word :
UNION
	Raw:WORD;
	Status:cNord_Status;
	
	
END_UNION
END_TYPE

// Burkert Library/uSensor_Status
TYPE uSensor_Status :
UNION
	iStatus:INT;
	eStatus:eSensor_Status;
END_UNION
END_TYPE

// Level_1/uAnalog_Pump_Modes
TYPE uAnalog_Pump_Modes :
UNION
	iMode:INT;
	eMode:eAnalog_Pump_Modes;
END_UNION
END_TYPE

// Level_1/uAnalog_Pump_Status
TYPE uAnalog_Pump_Status :
UNION
	iStatus:INT;
	eStatus:eAnalog_Pump_Status;
END_UNION
END_TYPE

// Level_1/uContactor_Modes
TYPE uContactor_Modes :
UNION
	iMode:INT;
	eMode:Contactor_Modes;
END_UNION
END_TYPE

// Level_1/uDI_Mode
TYPE uDI_Mode :
UNION
	iMode:INT;
	eMode:DI_Modes;
END_UNION
END_TYPE

// Level_1/uDI_Status
TYPE uDI_Status :
UNION
	iStatus:INT;
	eStatus:DI_Status;
END_UNION
END_TYPE

// Level_1/uDo_Modes
TYPE uDo_Modes :
UNION
	iMode:INT;
	eMode:Do_modes;
END_UNION
END_TYPE

// Level_1/uHOA_Mode
TYPE uHOA_Mode :
UNION
	iMode:INT;
	eMode:Burkert.eHOA_Modes;
END_UNION
END_TYPE

// Level_1/uM_Pump_Modes
TYPE uM_Pump_Modes :
UNION
	iMode:INT;
	eMode:eM_Pump_Modes;
END_UNION
END_TYPE

// Level_1/uM_Pump_Status
TYPE uM_Pump_Status :
UNION
	iStatus:INT;
	eStatus:eM_Pump_Status;
END_UNION
END_TYPE

// Level_1/uVFD_Mode
TYPE uVFD_Mode :
UNION
	iMode:INT;
	eMode:eVFD_Modes;
END_UNION
END_TYPE

// Level_1/uVFD_Status
TYPE uVFD_Status :
UNION
	iStatus:INT;
	eStatus:eVFD_Status;
END_UNION
END_TYPE

// Burkert Library/e_8681_Modes
{attribute 'qualified_only'}
//{attribute 'strict'}
TYPE Burkert.e_8681_Modes :
(
	Auto := 0,
	Disabled,
	Open,
	Upper_Drain,
	Lower_Drain
);
END_TYPE

// Burkert Library/eAODD_Modes
{attribute 'qualified_only'}
//{attribute 'strict'}
{attribute 'to_string'}
TYPE eAODD_Modes :
(
	Auto := 0,
	Disabled,
	Manual,
	Prime
);
END_TYPE

// Burkert Library/eB336x_Modes
{attribute 'qualified_only'}
//{attribute 'strict'}
TYPE eB336x_Modes :
(
		Auto := 0,
	Closed,
	Open,
	Manual_Pos,
	Config
);
END_TYPE

// Burkert Library/eConfig_startTune
{attribute 'qualified_only'}
//{attribute 'strict'}
TYPE eConfig_startTune :
(
	Complete := 0,
	Abort:=1,
	x_Tune:=2,
	p_Tune:=3,
	p_Lin:=4,
	a_Tune:=5,
	m_Clean:=7,
	mQC:=9
);
END_TYPE

// Burkert Library/eHOA_Modes
{attribute 'qualified_only'}
//{attribute 'strict'}
{attribute 'to_string'}
TYPE Burkert.eHOA_Modes :
(
	Off := 0,
	Auto,
	Manual
);
END_TYPE

// Burkert Library/LS_Modes
{attribute 'qualified_only'}
{attribute 'strict'}
TYPE LS_Modes :
(
	Active := 0,
	Forced_Off,
	Forced_On
);
END_TYPE

// Burkert Library/Positioner_Modes
{attribute 'qualified_only'}
{attribute 'strict'}
TYPE Positioner_Modes :
(
	Auto := 0,
	Manual_Open,
	Manual_Close,
	Manual_Position
);
END_TYPE

// Burkert Library/PT_Modes
{attribute 'qualified_only'}
//{attribute 'strict'}
TYPE PT_Modes :
(
	Active := 0,
	Forced,
	Alarms_Disabled,
	Alarm_Reset,
	OffLine
);
END_TYPE

// Burkert Library/Reset_Relay_Mode
{attribute 'qualified_only'}
{attribute 'strict'}
TYPE Reset_Relay_Mode :
(
	Off := 0,
	On
	
);
END_TYPE

// Level_1/eVFD_Modes
{attribute 'qualified_only'}
//{attribute 'strict'}
{attribute 'to_string'}
TYPE eVFD_Modes :
(
	Auto := 0,
	Disabled,
	Manual,
	Reset,
	Simulate:=10
);
END_TYPE

// eAnalog_Control_Modes
{attribute 'qualified_only'}
//{attribute 'strict'}
{attribute 'to_string'}
TYPE eAnalog_Control_Modes :
(
	Auto := 0,
	OFF,
	Manual
);
END_TYPE

// eFilter_Manager_Modes
{attribute 'qualified_only'}
{attribute 'strict'}
TYPE eFilter_Manager_Modes :
(
	Auto := 0,
	Filter_1,
	Filter_2
);
END_TYPE

// eFilter_Mode
{attribute 'qualified_only'}
{attribute 'strict'}
TYPE eFilter_Mode :
(
	Idle := 0,
	Prime,
	Active,
	Drain,
	Rinse,
	Disabled
);
END_TYPE

// eTempered_Modes
{attribute 'qualified_only'}
//{attribute 'strict'}
{attribute 'to_string'}
TYPE eTempered_Modes :
(
	Mix:=0,
	HW_Only,
	CW_Only
);
END_TYPE

// Level_3/eBrite_Modes
{attribute 'qualified_only'}
//{attribute 'strict'}
{attribute 'to_string'}
TYPE eBrite_Modes :
(
	Off := 0,
	ON//,
	//Crash
);
END_TYPE

// Level_3/eCLT_Modes
{attribute 'qualified_only'}
//{attribute 'strict'}
{attribute 'to_string'}
TYPE eCLT_Modes :
(
	Off := 0,
	Auto,
	Manual
	
);
END_TYPE

// Level_3/eFermenter_Modes
{attribute 'qualified_only'}
//{attribute 'strict'}
{attribute 'to_string'}
TYPE eFermenter_Modes :
(
	Off := 0,
	Ferment,
	Crash
);
END_TYPE

// Level_3/eGR_Modes
{attribute 'qualified_only'}
//{attribute 'strict'}
{attribute 'to_string'}
TYPE eGR_Modes :
(
	Off := 0,
	Mill,
	Transfer,
	Auto_Halt
	
);
END_TYPE

// Level_3/eHLT_Modes
{attribute 'qualified_only'}
//{attribute 'strict'}
{attribute 'to_string'}
TYPE eHLT_Modes :
(
	Off := 0,
	Auto,
	Manual
	
);
END_TYPE

// Level_3/eKT_Modes
{attribute 'qualified_only'}
//{attribute 'strict'}
{attribute 'to_string'}
TYPE eKT_Modes :
(
	Auto := 0,
	OFF,
	Manual
);
END_TYPE

// Level_3/eLT_Modes
{attribute 'qualified_only'}
//{attribute 'strict'}
{attribute 'to_string'}
TYPE eLT_Modes :
(
	Off := 0,
	Auto,
	Manual,
	Pause
	
);
END_TYPE

// Level_3/eMM_Modes
{attribute 'qualified_only'}
//{attribute 'strict'}
{attribute 'to_string'}
TYPE eMM_Modes :
(
	Off := 0,
	Auto,
	Manual
);
END_TYPE

// Level_3/eRCP_Mode
{attribute 'qualified_only'}
//{attribute 'strict'}
TYPE eRCP_Mode :
(
	Ready:= 0,
	Activate,
	Save,
	Copy,
	Paste,
	ReLoad,
	Push_To_MT,
	Push_To_LT,
	Push_To_KT,
	Push_To_WP,
	Pull_From_MT,
	Pull_From_LT,
	Pull_From_KT,
	Pull_From_WP
	
);
END_TYPE

// Level_3/eWP_Modes
{attribute 'qualified_only'}
//{attribute 'strict'}
{attribute 'to_string'}
TYPE eWP_Modes :
(
	Auto := 0,
	OFF,
	Manual
);
END_TYPE

// Level_3/FV_Modes
{attribute 'qualified_only'}
//{attribute 'strict'}
TYPE FV_Modes :
(
	Off := 0,
	Ferment,
	Dry_Hop,
	Crash
	
);
END_TYPE

// Level_3/HLT_Blending_Modes
{attribute 'qualified_only'}
//{attribute 'strict'}
TYPE HLT_Blending_Modes :
(
	Off := 0,
	Auto_Run,
	Auto_Paused,
	Auto_Halt
	
);
END_TYPE

// Level_3/KTWP_Modes
{attribute 'qualified_only'}
//{attribute 'strict'}
{attribute 'to_string'}
TYPE KTWP_Modes :
(
	Off := 0,
	Auto_Run,
	Auto_Paused,
	Auto_Halt
	
);
END_TYPE

// Level_1/Contactor_Status
{attribute 'qualified_only'}
{attribute 'to_string'}
TYPE Contactor_Status :
(
	OFF := 0,
	Auto_FWD,
	Auto_Rev,
	Manual_FWD,
	Manual_Rev,
	FWD_Limit,
	REV_Limit
);
END_TYPE

// Level_1/DI_Status
{attribute 'qualified_only'}
//{attribute 'strict'}
{attribute 'to_string'}
TYPE DI_Status :
(
	Normal_Signal_OFF := 0,
	Normal_Signal_Active,
	ALARM_Signal_ACTIVE,
	ALARM_Signal_LOST,
	Forced_On,
	Forced_OFF,
	Liquid_Detected,		//6
	No_Liquid_Detected,		//7
	Liquid_Detected_Alarm,	//8
	No_Liquid_Detected_Alarm,	//9
	
	End_Status:=99
);
END_TYPE

// Level_1/DO_Status
{attribute 'qualified_only'}
//{attribute 'strict'}
{attribute 'to_string'}
TYPE DO_Status :
(
	OFF := 0,
	On,
	Forced_OFF,
	Forced_ON,
	
	LOCKED_OUT:=6,
	Interlocked,
	OFFLINE
);
END_TYPE

// Level_1/eAnalog_Pump_Status
{attribute 'qualified_only'}
//{attribute 'strict'}
{attribute 'to_string'}
TYPE eAnalog_Pump_Status :
(
	IDLE := 0,
	Running,
	Disabled,
	Prime,
	Manual,
	Complete,
	LOCKED_OUT,				//
	Interlocked,		//
	Offline,
	Pump_Fault,
	Fault//
);
END_TYPE

// Level_1/eAODD_Status
{attribute 'qualified_only'}
//{attribute 'strict'}
TYPE eAODD_Status :
(
	Idle:=0,
	Disabled,
	Active,
	Complete
);
END_TYPE

// Level_1/eM_Pump_Status
{attribute 'qualified_only'}
{attribute 'strict'}
{attribute 'to_string'}
TYPE eM_Pump_Status :
(
	Idle := 0,
	Active,
	Disabled,
	Manual_Run,
	Prime_Active,
	
	
	LOCKED_OUT:=6,				//
	Interlocked,		//
	Offline
	
);
END_TYPE

// Level_1/eVFD_Status
{attribute 'qualified_only'}
//{attribute 'strict'}
{attribute 'to_string'}
TYPE eVFD_Status :
(
	READY:=0,	
	A_Running,				//
	Disabled,				//	
	M_Runing:=4,					//
	Ramping,				//			
			

				
	LOCKED_OUT:=6,				//
	Interlocked,		//
	Offline,
	Fault,
	Low_Voltage,  //10
	Safe_Torque_Off,
	No_Motor_Load_Detected,		//	12
	Low_Low_Current_Alarm,		//13		Sensor:1
	Low_Current_Warning,				//	Sensor:2
	High_Current_Warning,
	High_High_Current_Alarm			//	16
);
END_TYPE

// Level_1/VFD_Fault_Status
{attribute 'qualified_only'}
//{attribute 'strict'}
{attribute 'to_string'}
TYPE VFD_Fault_Status :
(
	enum_member := 0,
	Motor_Temperature:=16
	
);
END_TYPE

// Level_2/eCondensate_Status
{attribute 'qualified_only'}
{attribute 'to_string'}
TYPE eCondensate_Status :
(
	IDLE := 0,
	Stage_1,
	Stage_2,
	High_Warning,
	HIGH_Alarm,
	Level_Switch_Fault,
	Fault,
	Purge		//7
	
);
END_TYPE

// Level_2/eFilter_Manager_Status
{attribute 'qualified_only'}
{attribute 'strict'}
TYPE eFilter_Manager_Status :
(
	Idle := 0,
	Filter_1_Active,
	Filter_2_Active,
	Filter_1_Not_Ready,
	Filter_2_Not_Ready
);
END_TYPE

// Level_2/eFilter_Status
{attribute 'qualified_only'}
{attribute 'strict'}
TYPE eFilter_Status :
(
	IDLE := 0,
	In_Service,
	In_Backwash,
	Draining,
	Pressure_Warning,
	Preessure_Alarm
);
END_TYPE

// Vessels/eBrite_Status
{attribute 'qualified_only'}
//{attribute 'strict'}
{attribute 'to_string'}
TYPE eBrite_Status :
(
	Sensor_Fault := 0,
	Valve_Fault,
	Coolant_Fault,
	IDLE,		//3
	Regulating,	//4
	Spare_5,
	Low_Warning,
	High_Warning,
	Low_Alarm,
	High_Alarm
);
END_TYPE

// Vessels/eCLT_Status
{attribute 'qualified_only'}
//{attribute 'strict'}
{attribute 'to_string'}
TYPE eCLT_Status :
(
	OFF := 0,
	Filling,
	Cool_And_Fill,
	Active,
	Fault,
	Line_Chase_Reset_Flow_Meter,
	Line_Chase_Open_Valve,
	Line_Chase_Active,
	Line_Chase_Complete,
	//Low_Tank_Level,
	//High_Tank_Temperature,
	Cooling,
	OK,
	//Low_Level,
	//Low_Low_Level,
	
	Pump_Intake_Dry,
	
	Tank_High_High_Level_Switch_Alarm,
	Tank_High_High_Level_Alarm,
	Tank_High_Level_Warning,
	Tank_Low_Level_Warning,
	Tank_Low_Low_Level_Alarm,
	Tank_Level_Fault,
	
	Tank_High_High_Temperature_Alarm,
	Tank_High_Temperature_Warning,
	Tank_Low_Temperature_Warning,
	Tank_Low_Low_Temperature_Alarm,
	Tank_Temperature_Fault,
	
	HTX_Discharge_High_High_Temperature_Alarm,
	HTX_Discharge_High_Temperature_Warning,
	HTX_Discharge_Low_Temperature_Warning,
	HTX_Discharge_Low_Low_Temperature_Alarm,
	HTX_Discharge_Temperature_Fault,
	
	Discharge_Pressure_High_High_Alarm,
	Discharge_Pressure_High_Warning,
	Discharge_Pressure_Low_Warning,
	Discharge_Pressure_Low_Low_Alarm,
	Discharge_Pressure_Fault,
	
	Recirc_ACV_Not_Ready,
	Glycol_ACV_Not_Ready,
	Fill_BCV_Not_Ready,
	
	PID_Recirc_Not_Ready,
	PID_Temp_Not_Ready,
	
	Pump_Not_ready,
	
	
	
	
	
	End_CLT_Status
);
END_TYPE

// Vessels/eHLT_Status
{attribute 'qualified_only'}
//{attribute 'strict'}
{attribute 'to_string'}
TYPE eHLT_Status :
(
	OFF := 0,
	Filling,
	Fill_And_Heat,
	Heating,
	Holding,
	Ready,
	
	Active,
	Fault,
	
	Line_Chase_Reset_Flow_Meter,
	Line_Chase_Open_Valve,
	Line_Chase_Active,
	Line_Chase_Complete,
	Low_Tank_Level,
	Low_Tank_Temperature,
	
	Strike_HW_Not_Ready,
	Strike_CW_Not_Ready,
	Sparge_HW_Not_Ready,
	Sparge_CW_Not_Ready,
	HTX_Outlet_ACV_Not_Ready,
	HTX_Steam_Not_Ready,
	
	
	Mix_Pump_Not_Ready,
	Recirc_Pump_Not_Ready,
	
	
	
	Strike_FIT_Not_Ready,
	Sparge_FIT_Not_Ready,
	HTX_FIT_Not_Ready,
	
	CW_Fill_Not_Ready,
	Recirc_To_HTX_Not_Ready,
	SprayBall_Not_Ready,
	SW_Main_BCV_Not_Ready,
	
	
	PID_HTX_Not_Ready,
	PID_Recirc_Not_Ready,
	
	Temperature_Not_Ready,
	Temperature_High_High_Alarm,
	Temperature_High_Warning,
	Temperature_Low_Warning,
	Temperature_Low_Low_Alarm,
	
	Strike_TT_Not_Ready,
	Strike_TT_High_High_Alarm,
	Strike_TT_High_Warning,
	Strike_TT_Low_Warning,
	Strike_TT_Low_Low_Alarm,
	
	
	Sparge_TT_Not_Ready,
	Sparge_TT_High_High_Alarm,
	Sparge_TT_High_Warning,
	Sparge_TT_Low_Warning,
	Sparge_TT_Low_Low_Alarm,
	
	
	HTX_Outlet_TT_Not_Ready,
	HTX_Outlet_TT_High_High_Alarm,
	HTX_Outlet_TT_High_Warning,
	HTX_Outlet_TT_Low_Warning,
	HTX_Outlet_TT_Low_Low_Alarm,
	
	HTX_Inlet_TT_Not_Ready,
	HTX_Inlet_TT_High_High_Alarm,
	HTX_Inlet_TT_High_Warning,
	HTX_Inlet_TT_Low_Warning,
	HTX_Inlet_TT_Low_Low_Alarm,
	
	
	Mix_Pump_Pressure_Not_Ready,
	Mix_Pump_Pressure_High_High_Alarm,
	Mix_Pump_Pressure_High_Warning,
	Mix_Pump_Pressure_Low_Warning,
	Mix_Pump_Pressure_Low_Low_Alarm,
	
	Recirc_Pressure_Not_Ready,
	Recirc_Pressure_High_High_Alarm,
	Recirc_Pressure_High_Warning,
	Recirc_Pressure_Low_Warning,
	Recirc_Pressure_Low_Low_Alarm,
	
	Level_Not_Ready,
	Level_High_High_Alarm,
	Level_High_Warning,
	Level_Low_Warning,
	Level_Low_Low_Alarm,
	
	Pump_Intake_LSLL_Not_Ready,
	Pump_Intake_Empty,
	Tank_LSHH_Not_Ready,
	Tank_High_High_Level_Switch_Alarm,
	
	End_HLT_Status
);
END_TYPE

// Vessels/eKT_Status
{attribute 'qualified_only'}
//{attribute 'strict'}
{attribute 'to_string'}
TYPE eKT_Status :
(
	IDLE := 0,
	System_Check,
	Ready,
	Start,
	Active,
	Complete,
	
	PreHeat,
	PreHeat_Complete,
	Opening_Wort_In_Valves,
	Start_Rocket,
	Rocket_Boil,
	Jacket_Boil,
	
	Full_Boil_Start,
	Full_Boil,
	Full_Boil_Complete,
	
	Waiting_For_Wort,
	Recieving_Wort,
	Enable_Rocket,
	Rocket_Active,
	Wort_Transfer_Start,
	Wort_Transfer_Active,
	Wort_Transfer_Complete,
	
	Transfer_Flush_Validate,
	Transfer_Flush_Active,				//
	Transfer_Flush_Complete,
	
	Holding_Temperature,
	Whirlpool_Start,
	WhirlPool_Active,
	Whirlpool_Not_Ready,
	Rest,
	Select_Fermenter,
	Enable_Cast_Out,
	CastOut,
	CastOut_Chase_Start,
	CastOut_Chase_Active,
	Rocket_Prepare,
	Rocket_Open_Vent,
	Rocket_Flood,
	Rocket_Drain,
	Drain_Complete,
	Tank_Rinse_Prepare,
	
	
	
	
	
	
	
	//////////////Alarms////////////////////
	
	KT_Chase_Valve_Not_Ready,
	KT_CIP_Recirc_Valve_Not_Ready,
	Pump_Chase_Valve_Not_Ready,
	KT_Pump_Drain_BCV_Valve_Not_Ready,
	KT_Rocket_Condensate_Valve_Not_Ready,
	KT_Rocket_Cooling_Isolation_Not_Ready,
	KT_Rocket_Cooling_Return_Valve_Not_Ready,
	KT_Rocket_Drain_Not_Ready,
	KT_Rocket_Shell_Drain_Not_Ready,
	KT_Rocket_Steam_Isolation_Not_Ready,
	KT_Spray_Ball_Chase_Valve_Not_Ready,
	KT_Tank_Bottom_Valve_Not_Ready,
	KT_TO_WP_Valve_Not_Ready,
	KT_Lower_Jacket_Steam_Valve_Not_Ready,
	KT_Middle_Jacket_Steam_Valve_Not_Ready,
	KT_Recirc_Valve_Not_Ready,
	KT_Rocket_Cooling_Control_Valve_Not_Ready,
	KT_Rocket_Steam_Control_Valve_Not_Ready,
	KT_Upper_Jacket_Steam_Valve_Not_Ready,
	KT_Lower_Jacket_PID_Not_Ready,
	KT_Middle_Jacket_PID_Not_Ready,
	KT_Rocket_Cooling_PID_Not_Ready,
	KT_Rocket_Heating_PID_Not_Ready,
	KT_Upper_Jacket_PID_Not_Ready,
	KT_Discharge_Temperature_Not_Ready,
	KT_Rocket_Discharge_Temperature_Not_Ready,
	KT_Vesel_Temperature_Not_Ready,
	//KT_Agitator_Not_Ready,
	//KT_Discharge_Pump_Not_Ready,
	KT_Condensate_Return_Valve_Not_Ready,
	KT_Rocket_Condensate_Return_Valve_Not_Ready,
	//Waiting_For_Wort,
	Enable_Lower_Jacket,
	Enable_Middle_Jacket,
	Enable_Upper_Jacket,
	//Enable_Rocket,
	Rocket_Empty,
	Rocket_No_Flow,
	Discharge_Pump_Not_Ready,
	Agitator_Not_Ready,
	Discharge_Pump_Intake_Empty,
	Rocket_Condensate_Fault,
	Jacket_Condensate_Fault,
	Whirlpool_Not_In_Auto,
	Whirlpool_Not_Idle,
	Drain_Active,
	Wort_In_Enable_Rocket,
	Wort_In_Rocket,
	Rinse,
	Rinse_Complete,
	Rinse_Tangent,
	Rinse_High_Outlet,
	Rinse_Low_Outlet,
	Rinse_Tank,
	Drain_1,
	Drain_2,
	Drain_3
	
	
	
);
END_TYPE

// Vessels/eLT_Status
{attribute 'qualified_only'}
//{attribute 'strict'}
{attribute 'to_string'}
TYPE eLT_Status :
(
	IDLE := 0,
	Recipe_Copied,
	LauterTun_Check,
	LauterTun_Ready,
	Foundation_Water_Prepare,	
	Foundation_Water_Prepare_SW,						//
	Foundation_Water,	
	Foundation_Water_SW,		//
	Foundation_Water_Complete,
	Mash_In_Check,
	Mash_In_Ready,	//
	Mash_In_Active,					//
	Mash_In_Complete,
	
	Underlet_Validate,
	UnderLet_Ready,			//
	Underlet_Active,					//
	Underlet_Complete,			//
	Underlet_Resting,						//
	Underlet_Rest_Complete,
	Underlet_Agitate,

	Vorlauf_Validate,
	Vorlauf_Ready,
	Raise_Plough,
	Vorlauf_Active,				//
	Vorlauf_Complete,
	
	Transfer_Validate,
	Transfer_Ready,
	Clear_FloWave_Volume,
	Transfer_Active,
	Transfer_Complete,
		
	Transfer_Sparge_Validate,
	Transfer_Sparge_Ready,
	Transfer_Sparge_Start,					//
	Transfer_Sparge_Active,
	Sparge_Complete_Waiting_on_Transfer,
	Transfer_Complete_Waiting_on_Sparge,
	Transfer_Sparge_Complete,			//
	
	Transfer_Empty_Validate,
	Transfer_Empty_Ready,
	Transfer_Empty_Running,
	Transfer_Min_Time_Complete,
	Transfer_Empty_Complete,
		//			//
	Transfer_Flush_Validate,
	Transfer_Flush_Active,				//
	Transfer_Flush_Complete,
	
	Tank_Clean_Active,
	Tank_Clean_Complete,
	
	Rinse_Active,				//
	Rinse_Complete,
			//
	Drain,						//
	Drain_Complete,
	
	Grain_out_Active,
	Raise_Elevator,
	Lower_Plough,
	Open_Grain_Door,
	Active,
	Complete,
	CIP_Active,
	Systems_Check,


	Validate,
	Ready,
	Resting,

	Open_KT_Supply_Valve,
	Low_Air,
	Low_Steam,
	
	Low_Pressure,
	Low_Flow,
	
	
	
	
	Paused,
	Kettle_Not_In_Auto,
	Kettle_Not_Idle,
	
	PreHeat_Active,
	PreHeat_Complete,
	
	Vorlauf_Low_Flow,
	Grain_Out_Complete,
	
	Rinse_Tank,
	Rinse_Sprayball_A,
	Rinse_Sprayball_A_B,
	Rinse_Sprayball_B,
	Rinse_Sprayball_B_A,
	Rinse_Tank_Complete,
	Rinse_Grant,
	Rinse_Grant_Active,
	Rinse_Grant_Complete,
	Close_Grain_Door,
	Rinse_Underlet,
	Rinse_Underlet_Active,
	
	
	
	
	//////////Tests Status 
	
	
	
	SprayBall_1_Not_Ready,
	SprayBall_2_Not_Ready,
	SprayBall_SW_Not_Ready,
	CIP_Recirc_BCV_Not_Ready,
	Grant_SW_Not_Ready,
	CIP_To_Grant_Not_Ready,
	Pump_Drain_BCV_Not_Ready,
	Drain_BCV_Not_Ready,
	Grant_Bottom_Not_Ready,
	CIP_Grant_Bypass_Not_Ready,
	Pump_Intake_SW_Not_Ready,
	UnderLet_Not_Ready,
	
	Vorlauf_Not_Ready,
	Grant_To_Kettle_Not_Ready,
	Grant_Supply_Not_Ready,
	Condensate_Valve_Not_Ready,
	Jacket_Steam_Not_Ready,
	
	Pump_Not_Ready,
	Rake_Not_Ready,
	Elevator_Not_Ready,
	Rake_Fan_Not_Ready,
	Grain_Door_Not_Ready,
	Grain_Conveyor_Not_Ready,
	
	Discharge_Flow_Not_Ready,
	
	Pump_Intake_LS_Dry,
	Grain_Door_Open,
	Grain_Door_Closed,
	Elevator_Upper_LImit,
	Elevator_Lower_Limit,
	
	SG_Sensor_Not_Ready,
	Pump_Pressure_Not_Ready,
	Grant_Level_Not_Ready,
	Elevtaor_Position_Not_Ready,
	Tank_Temperature_Not_Ready,
	False_Bottom_Upper_Pressure_Not_Ready,
	False_Bottom_Lower_Pressure_Not_Ready,
	
	SG_Sensor_High_High_Alarm,
	Pump_Pressure_High_High_Alarm,
	Grant_Level_High_High_Alarm,
	Elevtaor_Position_High_High_Alarm,
	Tank_Temperature_High_High_Alarm,
	False_Bottom_Upper_Pressure_High_High_Alarm,
	False_Bottom_Lower_Pressure_High_High_Alarm,
	
	SG_Sensor_High_Warning,
	Pump_Pressure_High_Warning,
	Grant_Level_High_Warning,
	Elevtaor_Position_High_Warning,
	Tank_Temperature_High_Warning,
	False_Bottom_Upper_Pressure_High_Warning,
	False_Bottom_Lower_Pressure_High_Warning,
	
	SG_Sensor_Low_Warning,
	Pump_Pressure_Low_Warning,
	Grant_Level_Low_Warning,
	Elevtaor_Position_Low_Warning,
	Tank_Temperature_Low_Warning,
	False_Bottom_Upper_Pressure_Low_Warning,
	False_Bottom_Lower_Pressure_Low_Warning,
	
	SG_Sensor_Low_Low_Alarm,
	Pump_Pressure_Low_Low_Alarm,
	Grant_Level_Low_Low_Alarm,
	Elevtaor_Position_Low_Low_Alarm,
	Tank_Temperature_Low_Low_Alarm,
	False_Bottom_Upper_Pressure_Low_Low_Alarm,
	False_Bottom_Lower_Pressure_Low_Low_Alarm,
	
	
	
	
	
	Status_End
	

		
);
END_TYPE

// Vessels/eMM_Status
{attribute 'qualified_only'}
//{attribute 'strict'}
{attribute 'to_string'}
TYPE eMM_Status :
(
	IDLE := 0,
	Waiting_For_Brew_Confirmation,
	PreHeat_Validate,
	PreHeat_Ready,
	PreHeating_Vessel,
	PreHeat_Complete,
	Mash_In_Validate,
	Mash_In_Ready,
	Foundation_Water,
	Strike_Prepare,
	Grain_Dispense,
	Grain_Rinse,
	Mash_In_Complete,
	Heat_Profile_1_Active,
	Heat_Profile_1_Complete,
	Heat_Profile_2_Active,
	Heat_Profile_2_Complete,
	Heat_Profile_3_Active,
	Heat_Profile_3_Complete,
	Heat_Profile_4_Active,
	Mash_Out_Validate,
	Mash_Out_Ready,
	Waiting_to_Transfer,
	Open_Transfer_Valve,
	Transfer_1,
	Transfer_Rest_1,
	Transfer_2,
	Transfer_Rest_2,
	Transfer_3,
	Transfer_Complete,
	Transfer_Chase_Validate,
	Transfer_Chase_Ready,
	Transfer_Chase_Active,
	Transfer_Chase_Complete,
	Mash_Out_Complete,
	Tank_Rinse_Validate,
	Tank_Rinse_Ready,
	Tank_Rinse_Active,
	Tank_Rinse_Complete,
	Tank_Drain,
	Tank_Drain_Complete,
	MashOut_Heat,
	Heat_1_Rest,
	Heat_2_Rest,
	Heat_3_Rest,
	
	
	
	
	
	
	Low_Steam,
	Low_Air,
	Upper_Jacket_Not_In_Auto,
	Middle_Jacket_Not_In_Auto,
	Lower_Jacket_Not_In_Auto,
	Upper_Jacket_Valve_Not_In_Auto,
	Middle_Jacket_Valve_Not_In_Auto,
	Lower_Jacket_Valve_Not_In_Auto,
	Grain_Hopper_Valve_Not_In_Auto,
	Strike_Water_System_Not_Ready,
	
	LT_Not_In_Auto,
	LT_Grain_Door_Not_Closed,
	LT_Agitator_Not_Ready,
	LT_Rake_Not_Ready,
	LT_Pump_Not_Ready,
	LT_Sparge_Not_Ready,
	Line_Chase_Not_Available,
	LT_Not_Waiting_For_Mash,
	Rinse_Valve_A,
	Rinse_Valve_A_B,
	Rinse_Valve_B,
	Rinse_Valve_B_A,
	
	//Extra's added to accomadate MLT
	Vorlauf_Active,
	Vorlauf_Complete,
	Sparge_Active,
	Sparge_Complete,
	Underlet_Start,
	Underlet_Active,
	Underlet_Complete,
	Grain_Out,
	Grain_Out_Complete,
	Rinse_Grant,
	Rinse_Underlet,
	Rinse_Vessel,
	Underlet_Mix,
	Underlet_Rest,
	
	
	
	Lower_Steam_ACV_Not_Ready,
	Middle_Steam_ACV_Not_Ready,
	Upper_Steam_ACV_Not_Ready,
	Strike_HW_Not_Ready,
	Strike_CW_Not_Ready,
	
	Pump_Not_Ready,
	Agitator_Not_Ready,
	
	MM_Temp_Not_Ready,
	MM_Temp_High_High_Alarm,
	MM_Temp_High_Warning,
	MM_Temp_Low_Warning,
	MM_Temp_Low_Low_Alarm,
	
	Level_Not_Ready,
	Level_High_High_Alarm,
	Level_High_Warning,
	Level_Low_Warning,
	Level_Low_Low_Alarm,

	
	PID_Lower_Jacket_Not_Ready,
	PID_Middle_Jacket_Not_Ready,
	PID_Upper_Jacket_Not_Ready,
	
	Strike_BCV_Not_Ready,
	Tank_Bottom_BCV_Not_Ready,
	MM_to_LT_BCV_Not_Ready,
	SprayBall_Utility_BCV_Not_Ready,
	PumpSeal_BCV_Not_Ready,
	Drain_BCV_Not_Ready,
	SprayBall_1_BCV_Not_Ready,
	SprayBall_2_BCV_Not_Ready,
	Chase_BCV_Not_Ready,
	Pump_Intake_Dry,
	
	

	MM_Status_End
);
END_TYPE

// Vessels/eWP_Status
{attribute 'qualified_only'}
//{attribute 'strict'}
{attribute 'to_string'}
TYPE eWP_Status :
(
	IDLE := 0,
	Recipe_Copy,
	Ready_For_Wort,
	Whirpool_Validate,
	WhirlPool_Active,
	Whirpool_Complete,
	Ready,
	Running,
	Active,
	Profile_2,
	Profile_3,
	Cast_out_1,
	Profile_4,
	Resting,
	Rest_Complete,
	Select_Fermenter,
	Fermenter_Capacity_Error,
	CastOut_Validate,
	CastOut_Start,
	CastOut_Active,
	CastOut_Complete,
	Chase_Validate,
	Chase_Active,
	Chase_Complete,
	Rinse_Validate,
	Rinse_Active,
	Rinse_Complete,

	Pump_Not_Ready,
	Trub_Rinse_Validate,
	Trub_Rinse_active,
	Trub_Rinse_Drain,
	Trub_Rinse_Complete,
	Drain_Active,
	Drain_Complete,
	CIP_1_Fill,
	CIP_1_Active,
	CIP_1_Complete,
	CIP_2_Fill,
	CIP_2_Active,
	CIP_2_Complete
	
	
	
	
	
);
END_TYPE

// 95 Base Mappings/Level_0/IoLink_Mapping
{attribute 'qualified_only'}
{attribute 'to_string'}
TYPE IoLink_Mapping :
(
	Master_001 := 0,
	IoLink_End
);
END_TYPE

// 95 Base Mappings/Level_0/ME44AI_Mapping
{attribute 'qualified_only'}
{attribute 'to_string'}
TYPE ME44AI_Mapping :
(
	GW1_S1_AI := 0,
	
	ME44AI_End

);
END_TYPE

// 95 Base Mappings/Level_0/ME44AO_Mapping
{attribute 'qualified_only'}
{attribute 'to_string'}
TYPE ME44AO_Mapping :
(
	GW1_S1_AO := 0,
	
	
	ME44AO_End
);
END_TYPE

// 95 Base Mappings/Level_0/ME44DI_Mapping
{attribute 'qualified_only'}
{attribute 'to_string'}
TYPE ME44DI_Mapping :
(
	GW1_S1_DI := 0,
	
	ME44DI_End
);
END_TYPE

// 95 Base Mappings/Level_0/ME44DO_Mapping
{attribute 'qualified_only'}
{attribute 'to_string'}
TYPE ME44DO_Mapping :
(
	GW1_S1_DO := 0,
	
	
	ME44DO_End
);
END_TYPE

// 95 Base Mappings/Level_0/me64_Mapping
{attribute 'qualified_only'}
{attribute 'to_string'}
TYPE me64_Mapping :
(
	ME64_001 := 0,
	ME64_End

);
END_TYPE

// 95 Base Mappings/Level_1/ACV_Mapping_1
{attribute 'qualified_only'}
{attribute 'to_string'}
TYPE ACV_Mapping_1 :
(
	ACV_001_Analog:=0,	
	CW1,
	CW2,
	HW1,
	HW2,

	
	ACV_End
);
END_TYPE

// 95 Base Mappings/Level_1/AIT_Mapping_1
{attribute 'qualified_only'}
{attribute 'to_string'}
TYPE AIT_Mapping_1 :
(
	AIT_001 := 0,	
	AIT_002,			
	AIT_End
);
END_TYPE

// 95 Base Mappings/Level_1/b8653_mapping
{attribute 'qualified_only'}
{attribute 'to_string'}
TYPE b8653_mapping :
(
	PM_001 := 0,
	b8653_End
);
END_TYPE

// 95 Base Mappings/Level_1/BCV_Mapping_1
{attribute 'qualified_only'}
{attribute 'to_string'}
TYPE BCV_Mapping_1 :
(
	BCV_001_IO := 0,	

	
	 
	BCV_END
);
END_TYPE

// 95 Base Mappings/Level_1/cSensor_Mapping
{attribute 'qualified_only'}
{attribute 'to_string'}
TYPE cSensor_Mapping :
(
	FV_001 := 0,
	FV_002,
	FV_003,
	
	BBT001,
	
	
	cSensor_End
	
);
END_TYPE

// 95 Base Mappings/Level_1/dACV_Mapping
{attribute 'qualified_only'}
{attribute 'to_string'}
TYPE dACV_Mapping :
(
	ACV_001_Digital:=0,	
	FV001_Top,			
	FV001_Middle,		
	FV001_Bottom,		
	
	ACV_End
);
END_TYPE

// 95 Base Mappings/Level_1/dBCV_Mapping
{attribute 'qualified_only'}
{attribute 'to_string'}
TYPE dBCV_Mapping :
(
	BCV_001_eDip := 0,	 
	BCV_002_CanOpen,
	BCV_003_IoLink,
	BCV_004_ModbusTCP,
	BCV_005_Profinet,
	BCV_006_EtherCat,
	
	FV001_Top,			
	FV001_Middle,		
	FV001_Bottom,	

	
	BCV_END
);
END_TYPE

// 95 Base Mappings/Level_1/DI_Mapping
{attribute 'qualified_only'}
{attribute 'to_string'}
TYPE DI_Mapping :
(
	BCV_001_Lim_1:=0,
	BCV_001_Lim_2,
	DI_end
);
END_TYPE

// 95 Base Mappings/Level_1/Do_Mapping
{attribute 'qualified_only'}
{attribute 'to_string'}
TYPE Do_Mapping :
(
	BCV_001_CMD:=0,
	DO_001,
	AP_001_FWD,
	AP_001_Rev,
	
	Do_End
);
END_TYPE

// 95 Base Mappings/Level_1/FIT_Mapping_1
{attribute 'qualified_only'}
{attribute 'to_string'}
TYPE FIT_Mapping_1 :
(
	FIT_001_Hz:=0,			
	FIT_002_Count,		
	FIT_003_Dual,
	FIT_004_Digital,	
	HW_FIT,
	CW_FIT,
	

	
	
	
	
	
	
	
	FIT_End
);
END_TYPE

// 95 Base Mappings/Level_1/LS_Mapping_1
{attribute 'qualified_only'}
{attribute 'to_string'}
TYPE LS_Mapping_1 :
(
	LSLL_001:=0,
	LSLL_002,
	LSHH_003,
	LSHH_004,
	LSLL_005,
	
	
	LS_End
);
END_TYPE

// 95 Base Mappings/Level_1/PT_Mapping_1
{attribute 'qualified_only'}
{attribute 'to_string'}
TYPE PT_Mapping_1 :
(
	PT_101:=0,
	Mix_PT,
	PT_End
);
END_TYPE

// 95 Base Mappings/Level_1/s8050_Mapping
{attribute 'qualified_only'}
{attribute 'to_string'}
TYPE s8050_Mapping :
(
	FIT_001 := 0,

	
	
	
	
	s8050_End
	
);
END_TYPE

// 95 Base Mappings/Level_1/s8228_Mapping
{attribute 'qualified_only'}
{attribute 'to_string'}
TYPE s8228_Mapping :
(
	CND_001:=0,
	

	s8228_End
);
END_TYPE

// 95 Base Mappings/Level_1/s8312_Mapping
{attribute 'qualified_only'}
{attribute 'to_string'}

//8312 Pressure
TYPE s8312_Mapping :
(
	PT_001:=0,
	HW_Inlet,
	HW_outlet,
	CW_Inlet,
	CW_outlet,
						
	
	
	
	
	S8312_End
);
END_TYPE

// 95 Base Mappings/Level_1/s8412_Mapping
{attribute 'qualified_only'}
{attribute 'to_string'}

//8312 Temperature
TYPE s8412_Mapping :
(
	TT_001:=0,
	
	
	
	
	
	s8412_End
);
END_TYPE

// 95 Base Mappings/Level_1/SV_Mapping
{attribute 'qualified_only'}
{attribute 'to_string'}
TYPE SV_Mapping :
(
	SV_001:=0,
	
	
	SV_END
);
END_TYPE

// 95 Base Mappings/Level_1/TT_Mapping_1
{attribute 'qualified_only'}
{attribute 'to_string'}
TYPE TT_Mapping_1 :
(
	TT_101:=0,
	
	FV001_Top,		
	FV001_Middle,	
	FV001_Bottom,	
	
	HW_Supply_TT,
	CW_Supply_TT,
	Mix_TT,
	TT_End
);
END_TYPE

// 95 Base Mappings/Level_1/v336x_Mapping
{attribute 'qualified_only'}
{attribute 'to_string'}
TYPE v336x_Mapping :
(
	v336x_001:=0,			

	
	v3363_End
);
END_TYPE

// 95 Base Mappings/Level_2/Analog_Pump_Mapping
{attribute 'qualified_only'}
{attribute 'to_string'}
TYPE Analog_Pump_Mapping :
(
	AP_001 := 0,

	
	Analog_Pump_End
);
END_TYPE

// 95 Base Mappings/Level_2/mPump_Mapping
{attribute 'qualified_only'}
{attribute 'to_string'}
TYPE mPump_Mapping :
(
	mPump_001 := 0,
	mPump_End
);
END_TYPE

// 95 Base Mappings/Level_2/PID_Mapping_1
{attribute 'qualified_only'}
{attribute 'to_string'}
TYPE PID_Mapping_1 :
(
	PID_001:=0,
	HW_PID,
	CW_PID,
	Mix,
	FV_001,
	FV_002,
	FV_003,
	
	
	BBT001,
	
	PID_End
);
END_TYPE

// 95 Base Mappings/Level_2/Stack_Light_Mapping
{attribute 'qualified_only'}
{attribute 'to_string'}
TYPE Stack_Light_Mapping :
(
	Light_001 := 0,
	
	
	Stack_Light_End
	
);
END_TYPE

// 95 Base Mappings/Level_2/VFD_Mapping
{attribute 'qualified_only'}
{attribute 'to_string'}
TYPE VFD_Mapping :
(
	VFD_001 := 0,	

	
	Eaton_VFD_End
);
END_TYPE

// 95 Base Mappings/Level_3/Alarm_Offset_Mapping
{attribute 'qualified_only'}
{attribute 'to_string'}
TYPE Alarm_Offset_Mapping :
(
	HWT := 0,
	CWT,
	TT_101,
	Head_Pressure,
	Filter_1,
	Filter_2,
	
	Alarm_Offset_End
);
END_TYPE

// 95 Base Mappings/Level_3/Brite_Mapping_1
{attribute 'qualified_only'}
{attribute 'to_string'}
TYPE Brite_Mapping_1 :
(
	BBT001 := 0,

	Brite_End
	
);
END_TYPE

// 95 Base Mappings/Level_3/Fermenter_Mapping_1
{attribute 'qualified_only'}
{attribute 'to_string'}
TYPE Fermenter_Mapping_1 :
(
	FV001 := 0,
	FV002,
	FV003,

	Fermenter_End
	
);
END_TYPE

// Level_1/HMI_Analog_Pump
TYPE HMI_Analog_Pump EXTENDS cAnalog_Pump :
STRUCT
	strName:STRING;
	strMode:STRING;
	strStatus:STRING;
END_STRUCT
END_TYPE

// Level_1/HMI_Contactor_DUT
TYPE HMI_Contactor_DUT EXTENDS cContactor :
STRUCT
	strName:STRING;
	strMode:STRING;
	strStatus:STRING;
END_STRUCT
END_TYPE

// Level_1/HMI_M_Pump
TYPE HMI_M_Pump EXTENDS cM_Pump :
STRUCT
	strName:STRING;
	strMode:STRING;
	strStatus:STRING;
END_STRUCT
END_TYPE

// Level_1/HMI_VFD_Eaton_DUT
TYPE HMI_VFD_Eaton_DUT EXTENDS cVFD_Eaton_DUT :
STRUCT
	strName:STRING;
	strMode:STRING;
	strStatus:STRING;
END_STRUCT
END_TYPE

// Level_2/HMI_PID
TYPE HMI_PID EXTENDS cPID_DUT :
STRUCT
	strName:STRING;
	strMode:STRING;
	strStatus:STRING;
END_STRUCT
END_TYPE

// Level_3/HMI_Brite
TYPE HMI_Brite EXTENDS cBrite_DUT :
STRUCT
	strName:STRING;
END_STRUCT
END_TYPE

// Level_3/HMI_Fermenter
TYPE HMI_Fermenter EXTENDS cFermenter_DUT :
STRUCT
	strName:STRING[30];
	//strMode:STRING[30];
	//strStatus:STRING[80];
END_STRUCT
END_TYPE

// In Burkert Device Library/Base_Declarations/cBase_FIT
TYPE cBase_FIT :
STRUCT
	Rate:Burkert.Burkert.cAIT;
	Total:REAL;
	PLC_Reset:BOOL;
	//Counts	:	UDINT;
	//Frequency	:REAL;
	K:REAL;
	HMI_Reset:BOOL;
END_STRUCT
END_TYPE

// In Burkert Device Library/LeveL_1/cACV
TYPE Burkert.cACV :
STRUCT
	HMI_CMD:REAL;
	PLC_CMD:REAL;
	Valve_Actual:REAL;

	Mode:uACV_Mode;//Burkert.eACV_Modes;
	Status:uACV_Status;
	Ready:BOOL;

END_STRUCT
END_TYPE

// In Burkert Device Library/LeveL_1/cAIT
TYPE Burkert.cAIT EXTENDS Burkert.Burkert.cAIT :
STRUCT
	
	Analog_Scale	:	Analog_scale;
	Mode			:	uAIT_Mode;
	PCT_Scale:REAL;
END_STRUCT
END_TYPE

// In Burkert Device Library/LeveL_1/cAnalog_Sensor
TYPE Burkert.Burkert.cAIT :
STRUCT
	Burkert.cAlarm_Config	:	Burkert.cAlarm_Config;
	EU:		REAL;
	Ready:BOOL;
	Status:uSensor_Status;
	
END_STRUCT
END_TYPE

// In Burkert Device Library/LeveL_1/cBCV
TYPE Burkert.cBCV :
STRUCT
	Mode	:uBCV_MODE;
	PLC_CMD	:	BOOL;
	Status:eBCV_Status;
	Ready:BOOL;

		
END_STRUCT
END_TYPE

// In Burkert Device Library/LeveL_1/cFIT
TYPE Burkert.cFIT EXTENDS cBase_FIT :
STRUCT

	Counts	:	UDINT;
	Frequency	:REAL;

END_STRUCT
END_TYPE

// In Burkert Device Library/LeveL_1/SV_DUT
TYPE SV_DUT :
STRUCT
	Mode:uBCV_Mode;
	Status:eBCV_Status;
	Q:BOOL;
	PLC_CMD:BOOL;
	Ready:BOOL;
	Namur:uNamur;
	strNamur:STRING[30];
END_STRUCT
END_TYPE

// In Burkert Device Library/To be Sorted/ACV_eDip
TYPE ACV_eDip :
STRUCT
	DirChanges:REAL;
	TravelAccu:REAL;
	XTunes:UINT;
	DeviceSupplyVoltage:REAL;
	DeviceTemperature:REAL;
	IdentNumber:UDINT;
	currOPmode:BYTE;
	ProductCode:UDINT;
	SerialNumber:UDINT;
	DEVmax:REAL;
	POSmonitor_Error:BYTE;
	currTUNEstatus:BYTE;
	Valve_Status:BYTE;
	
	
	
END_STRUCT
END_TYPE

// In Burkert Device Library/To be Sorted/Alarm_Config
TYPE Burkert.cAlarm_Config :
STRUCT
	Hi_Hi_Alarm		:		REAL;
	Hi_Warn			:		REAL;
	Low_warn		:		REAL;
	Low_Low_Alarm	:	REAL;
	Silence:		BOOL;
	Debounce:		UINT;
	PCT_Alarm:		REAL;
	
END_STRUCT
END_TYPE

// In Burkert Device Library/To be Sorted/Alarm_Window
TYPE Alarm_Window :
STRUCT
	Target:REAL;
	Warn_Window:REAL;
	Alarm_Window:REAL;
	Alarm_Delay:UINT;
END_STRUCT
END_TYPE

// In Burkert Device Library/To be Sorted/Analog_scale
TYPE Analog_scale :
STRUCT
	Raw	:	REAL;
	Eu_Min	:	REAL 	:=0;
	Eu_Max	:	REAL 	:=100;
	Raw_Min	:	REAL 	:=4;
	Raw_Max	:	REAL	:=20;
	Override_Value	:	REAL;
	//Override	:BOOL;
	
		
END_STRUCT
END_TYPE

// In Burkert Device Library/To be Sorted/AODD_DUT
TYPE AODD_DUT :
STRUCT
	Base_Rate:REAL:=25;
	HMI_Target_Volume:REAL;
	HMI_Target_Rate:REAL;
	PLC_Target_Volume:REAL;
	PLC_Target_Rate:REAL;
	Duty_Cycle:REAL;
	Min_On_Seconds:INT:=10;
	Min_OFF_Seconds:INT:=2;
	Shots_Remaining:INT:=0;
	On_Time:REAL;
	Off_Time:REAL;
	Volume_Delivered:REAL;
	PLC_Run:BOOL;
	Mode:eAODD_Modes;
	Status:eAODD_Status;
END_STRUCT
END_TYPE

// In Burkert Device Library/To be Sorted/Asi_Node_DUT
TYPE Asi_Node_DUT :
STRUCT
	Detected:BOOL;
	PROJECTED:BOOL;
	Active:BOOL;
	Fault:BOOL;
	Analog_RX_0:WORD;
	Analog_RX_1:WORD;
	Analog_TX_0:WORD;
	Analog_TX_1:WORD;
	Digital_RX:BYTE;
	Digital_TX:BYTE;
	
	
END_STRUCT
END_TYPE

// In Burkert Device Library/To be Sorted/b8619_CND_DUT
TYPE b8619_CND_DUT :
STRUCT
	
ID_Revision:BYTE;
ID_Version:BYTE;
ID_Slot:BYTE;
ID_Type:BYTE;

Status_Link_Lost:BOOL;
Status_Calibration_Lost:BOOL;
Status_UserData_lost:BOOL;
Status_Factory_Data_Lost:BOOL;
Status_Clock_Faulty:BOOL;
Status_Probe_Error:BOOL;
Status_Probe_Warning:BOOL;
Status_Probe_Calibration:BOOL;
Status_Presence:BOOL;

Temp_Status:WORD;
CND_Status:WORD;
RTD:REAL;
Temperature:REAL;
Conductivity:REAL;
Resistivity:REAL;
TDS:REAL;
Concentration:REAL;

END_STRUCT
END_TYPE

// In Burkert Device Library/To be Sorted/b8619_Inputs_DUT
TYPE b8619_Inputs_DUT :
STRUCT
	ID_Revision:BYTE;
	ID_Version:BYTE;
	ID_Slot:BYTE;
	ID_Type:BYTE;
	Status_Link_Lost:BOOL;
	Status_Calibration_Lost:BOOL;
	Status_UserData_lost:BOOL;
	Status_Factory_Data_Lost:BOOL;
	Status_time_lost:BOOL;
	Status_Warning:BOOL;
	Status_Memory_Issue:BOOL;
	Status_Presence:BOOL;
	
	DI1_Status:WORD;
	DI2_Status:WORD;
	AI1_Status:WORD;
	AI2_Status:WORD;
	
	DI1_Hz:REAL;
	DI1_Flow:REAL;
	DI1_Total_A:REAL;
	DI1_Total_B:REAL;
	DI2_Hz:REAL;
	DI2_Flow:REAL;
	DI2_Total_A:REAL;
	DI2_Total_B:REAL;
	
	AI1_Raw:REAL;
	AI1_EU:REAL;
	AI2_Raw:REAL;
	AI2_EU:REAL;
	
	
END_STRUCT
END_TYPE

// In Burkert Device Library/To be Sorted/b8619_Main_DUT
TYPE b8619_Main_DUT :
STRUCT
	ID_Revision:BYTE;
	ID_Version:BYTE;
	ID_Slot:BYTE;
	ID_Type:BYTE;
	Status_Link_Lost:BOOL;
	Status_Calibration_Lost:BOOL;
	Status_UserData_lost:BOOL;
	Status_Factory_Data_Lost:BOOL;
	Status_time_lost:BOOL;
	Status_Warning:BOOL;
	Status_Memory_Issue:BOOL;
	Status_Presence:BOOL;
	
	M1_M3_Status:WORD;
	M4_M6_Status:WORD;
	System_Switch:WORD;
	DI1_Status:WORD;
	DI2_Status:WORD;
	DO1:WORD;
	DO2:WORD;
	AO1:REAL;
	AO2:REAL;
	DI1_Hz:REAL;
	DI1_Flow:REAL;
	DI1_Total_A:REAL;
	DI1_Total_B:REAL;
	DI2_Hz:REAL;
	DI2_Flow:REAL;
	DI2_Total_A:REAL;
	DI2_Total_B:REAL;
	
	
	
	
END_STRUCT
END_TYPE

// In Burkert Device Library/To be Sorted/b8619_PH_DUT
TYPE b8619_PH_DUT :
STRUCT
	ID_Revision:BYTE;
	ID_Version:BYTE;
	ID_Slot:BYTE;
	ID_Type:BYTE;
	
	Status_Link_Lost:BOOL;
	Status_Calibration_Lost:BOOL;
	Status_UserData_lost:BOOL;
	Status_Factory_Data_Lost:BOOL;
	Status_Clock_Faulty:BOOL;
	Status_Probe_Error:BOOL;
	Status_Probe_Warning:BOOL;
	Status_Probe_Calibration:BOOL;
	Status_Presence:BOOL;
	
	Temp_Status:WORD;
	PH_Status:WORD;
	RTD:REAL;
	Temperature:REAL;
	mv_PH:REAL;
	mv_ORP:REAL;
	PH:REAL;
	Impedance_Glass:REAL;
	Impedance_Ref:REAL;

END_STRUCT
END_TYPE

// In Burkert Device Library/To be Sorted/B8691_Asi_DUT
TYPE Burkert.B8691_Asi_DUT :
STRUCT
	Mode	:	Burkert.e_8681_Modes;
	Status	:	WORD;
	HMI_CMD	:	INT;
	PLC_CMD	:	INT;
	Status1 :eB8681_Status;
	Valve_Status:BYTE;
END_STRUCT
END_TYPE

// In Burkert Device Library/To be Sorted/c8694_PDin
TYPE c8694_PDin :
STRUCT
	Valve_Position:REAL;
	Target_Position:REAL;
	Namur_Status:e8691_Namur_Status;
	Valve_Status:e8691_Valve_Status;
	Open_Limit:BOOL;
	Close_Limit:BOOL;
	
END_STRUCT
END_TYPE

// In Burkert Device Library/To be Sorted/cFLOWave_DUT
TYPE cFLOWave_DUT :
STRUCT
	


	Acoustic_Trans:REAL;
	AcousticImpedance:REAL;
	Concentration_1:REAL;
	Concentration_2:REAL;
	Density:REAL;
	Density_Factor:REAL;;
	Dynamic_Viscosity:REAL;
	FoulingFactor:REAL;
	Gas_Bubble_Factor:REAL;
	Kinematic_vicosity:REAL;
	Liquid_Velocity:REAL;
	Mass_Flow:REAL;
	Mass_Total_1:REAL;
	Mass_Total_2:REAL;	
	Namur_Status:INT;
	Saw_Group_Velocity:REAL;
	SpeedOfSound:REAL;
	Temp:REAL;
	Total_1:REAL;
	Total_2:REAL;
	Turbulance_Factor:REAL;
	Viscosity_Factor:REAL;
	Volume_Flow:REAL;	
	FIT_1:Burkert.cFIT;
	FIT_2:Burkert.cFIT;
	Status:eFloWave_Status;
	M_Reset_1:BOOL;
	M_Reset_2:BOOL;
	Burkert.cAlarm_Config:ARRAY[0..3] OF Burkert.cAlarm_Config;
	Locate:BOOL;
	Maintenance:BOOL;
END_STRUCT
END_TYPE

// In Burkert Device Library/To be Sorted/CND_8619
TYPE CND_8619 :
STRUCT
	RTD_OHM:REAL;
	Temperature:REAL;
	Conductivity:REAL;
	Resistivity:REAL;
	TDS:REAL;
	Concentration:REAL;
END_STRUCT
END_TYPE

// In Burkert Device Library/To be Sorted/cSDO_DUT
TYPE cSDO_DUT :
STRUCT
	NodeId:BYTE;
	Index:WORD;
	SubIndex:BYTE;
	Bytes:WORD;
	Data:ARRAY[0..3] OF BYTE;
	Read:BOOL;
	Write:BOOL;
	Done:BOOL;
	Busy:BOOL;
	Error:BOOL;
	
	
END_STRUCT
END_TYPE

// In Burkert Device Library/To be Sorted/eDip_8681_DUT
TYPE eDip_8681_DUT :
STRUCT
	Outputs:ARRAY[0..3] OF BOOL;
	Inputs:ARRAY[0..3] OF BOOL;
	Position:REAL;
	Namur:BYTE;
	Status1:eB8681_Status;
	PLC_CMD:INT;
	HMI_CMD:INT;
	Mode:INT;	
END_STRUCT
END_TYPE

// In Burkert Device Library/To be Sorted/eDip_DDO
TYPE eDip_DDO :
STRUCT
	Ident:UDINT; //16#2000-2
	Serial:UDINT; //16#2000-7
	Product_Code:UDINT;//16#2000-8
	Manufacture_DATE:UDINT; //16#2000-3
END_STRUCT
END_TYPE

// In Burkert Device Library/To be Sorted/eDip_DSO
TYPE eDip_DSO :
STRUCT
	NamurNe107:BYTE;//16#2004-1
	Temperature:REAL; //16#2004-2
	Voltage:REAL;//16#2004-3
	Operational_Time_S:UDINT;//16#2004-4
	Max_Temp:REAL;//16#2004-5
	Min_Temp:REAL;//16#2004-6
	Max_Voltage:REAL;//16#2004-7
	Min_Voltage:REAL;//16#2004-8
END_STRUCT
END_TYPE

// In Burkert Device Library/To be Sorted/eDip_MFC_DUT
TYPE eDip_MFC_DUT :
STRUCT
	
	ActualFlow:REAL;
	ActuatingVariable:REAL;
	MediumTemperature:REAL;
	Totalizer:REAL;
	UsedSetPooint:REAL;
	SetPoint:REAL;
	CurrentDutyCycle:REAL;
	NamurStatus:BYTE;
	
	
	Mode:INT;
	PLC_SP:REAL;
	HMI_SP:REAL;
	Locate:BOOL;
	Maintenance:BOOL;
	
	
END_STRUCT
END_TYPE

// In Burkert Device Library/To be Sorted/FV_DUT
TYPE FV_DUT :
STRUCT
	Mode:INT;

	Ferment_Setpoint:REAL;
	Dry_Hop_Setpoint:REAL;
	Crash_Setpoint:REAL;
	
		
		
END_STRUCT
END_TYPE

// In Burkert Device Library/To be Sorted/HLT_Blending_DUT
TYPE HLT_Blending_DUT :
STRUCT
	Mode:INT;
	Mode_Name:eHLT_Modes;
	
	Command:INT;
	Command_Ind:ARRAY [0..20] OF INT;
	Command_Name:HLT_Blending_Steps;
	Command_Reset:TON;
		
	Step_Complete:INT;
	Step_Complete_Reset:TON;
		
	Status:INT;

	Step:INT;
	Step_Memory:INT;
	Step_Memory_Name:HLT_Blending_Steps;
	
	Step_Bits:ARRAY [0..20] OF BOOL;

	Current_Step_Setpoint:DINT;
	Current_Step_Accumulated:DINT;
	
	Flow_Count_Step:BOOL;
	Time_Count_Step:BOOL;
	Step_Done:BOOL;
	
	Setpoint:ARRAY [0..20] OF INT;
	Rate_Setpoint:ARRAY [0..20] OF REAL;

	MM_HW_PID:PID_DUT;
	MM_CW_PID:PID_DUT;
	LT_HW_PID:PID_DUT;
	LT_CW_PID:PID_DUT;
		
	Max_Pressure_Set:REAL;
	
	Alarms:DINT;
	Alarm_Present:BOOL;
	Alarms_Display:DINT;
	Alarm_Display_Index:DINT;
	Alarm_Reset:DINT;
	
	Auto_Mode_Req:INT;
		
END_STRUCT
END_TYPE

// In Burkert Device Library/To be Sorted/HLT_Chase_DUT
TYPE HLT_Chase_DUT :
STRUCT
	Target:eHLT_Chase_Targets;
	Volume:REAL;
	Rate:REAL;
END_STRUCT
END_TYPE

// In Burkert Device Library/To be Sorted/PH_8619
TYPE PH_8619 :
STRUCT
	RTD_OHM:REAL;
	Temperature:REAL;
	mv:REAL;
	ORP:REAL;
	PH:REAL;
	
	
END_STRUCT
END_TYPE

// In Burkert Device Library/To be Sorted/PT_Config_DUT
TYPE PT_Config_DUT :
STRUCT
	Burkert.cAlarm_Config	:	Burkert.cAlarm_Config;
	Analog_Scale	:	Analog_scale;
	Mode			:	PT_Modes;
	
END_STRUCT
END_TYPE

// In Burkert Device Library/To be Sorted/SDO
TYPE SDO :
STRUCT
	Index:WORD;
	Node:BYTE;
	SubIndex:BYTE;
END_STRUCT
END_TYPE

// In Burkert Device Library/To be Sorted/Steam_Set_Config_DUT
TYPE Steam_Set_Config_DUT :
STRUCT
	Isolation_Open_Demand:REAL;
	Isolation_CLose_Demand:REAL;
	ACV_Config:Burkert.cACV;
	BV_Config:Burkert.cBCV;
	
	
END_STRUCT
END_TYPE

// In Burkert Device Library/To be Sorted/Steam_Set_DUT
TYPE Steam_Set_DUT :
STRUCT
	Mode:UINT;
	Status:UINT;
	ACV:Burkert.cACV;
	BV:Burkert.cBCV;
END_STRUCT
END_TYPE

// In Burkert Device Library/To be Sorted/TT_Config_DUT
TYPE TT_Config_DUT :
STRUCT
	Burkert.cAlarm_Config	:	Burkert.cAlarm_Config;
	Analog_Scale	:	Analog_scale;
	Mode			:	Burkert.TT_Modes;
	
END_STRUCT
END_TYPE

// In Burkert Device Library/To be Sorted/Vessel_Config_Dut
TYPE Vessel_Config_Dut :
STRUCT
	MODE:INT;
	Batch_ID:INT;
	Target_Time_minutes:UINT;
	Base_SP:REAL;
	Alarms:Burkert.cAlarm_Config;
	DT_Rate_C_Min:REAL;
	Zone_Temp_offset:REAL:=0.5;
	
END_STRUCT
END_TYPE

// In Burkert Device Library/To be Sorted/Word_as_Real_DUT
TYPE Word_as_Real_DUT :
UNION
	Words:ARRAY[0..1] OF WORD;
	rReal:REAL;
END_UNION
END_TYPE

// Level_0/Adam_6050/cAdam_6050_MBTCP
TYPE cAdam_6050_MBTCP :
STRUCT
	Raw_DI:DWORD;		//40301
	Raw_DO:DWORD;		//40303
	Counter_Values:ARRAY[0..11] OF DWORD;		//40001-40024
	Counter_Control:ARRAY[0..11] OF cAdam_6050_Control;		//0x32 24 4 bytes
	
	
END_STRUCT
END_TYPE

// Level_0/Adam_6052/cAdam_6052_Control
TYPE cAdam_6052_Control :
STRUCT
	Enable:WORD;
	Clear:WORD;
	Clear_Overflow:WORD;
	Latch_Status:WORD;
	
END_STRUCT
END_TYPE

// Level_0/Adam_6052/cAdam_6052_MBTCP
TYPE cAdam_6052_MBTCP :
STRUCT
	Raw_DI:DWORD;		//40301
	Raw_DO:DWORD;		//40303
	Counter_Values:ARRAY[0..7] OF DWORD;		//40001-40024
	Counter_Control:ARRAY[0..7] OF cAdam_6052_Control;			//0x32 24 3 bytes
	
	
END_STRUCT
END_TYPE

// Level_0/IO-Link/c8694_Io_Link
TYPE c8694_Io_Link :
STRUCT
	HMI_CMD:REAL;
	PLC_CMD:REAL;
	Valve_Actual:REAL;
	Mode:Burkert.eACV_Modes;
	Status:ACV_Status;
	IOLink_PDin:c8694_Pdin;
	IoLink_Diag:c8694_IoLink_Diag;
	IoLink_Command:e8694_IoLink_Commands;
	xTune_Status:e8694_xTune_Status;
END_STRUCT
END_TYPE

// Level_0/IO-Link/cIFM_AL1340
TYPE cIFM_AL1340 :
STRUCT
	Port_1_RX:ARRAY[0..15] OF WORD;
	Port_2_RX:ARRAY[0..15] OF WORD;
	Port_3_RX:ARRAY[0..15] OF WORD;
	Port_4_RX:ARRAY[0..15] OF WORD;
	
	Port_1_TX:ARRAY[0..15] OF WORD;
	Port_2_TX:ARRAY[0..15] OF WORD;
	Port_3_TX:ARRAY[0..15] OF WORD;
	Port_4_TX:ARRAY[0..15] OF WORD;

	Port_Request:ARRAY[1..4] OF 	cIFM_AL1342_Acyclic_Request;
	Port_Response:ARRAY[1..4] OF cIFM_AL1342_Acyclic_Response;
	
	Request:cIFM_AL1342_Acyclic_Request;
	Response:cIFM_AL1342_Acyclic_Response;
	Acyclic_Request:BOOL;
	
	
	
	
	(*
	Port_Request:ARRAY[1..8] OF 	cIFM_AL1342_Acyclic_Request;
	Port_Response:ARRAY[1..8] OF cIFM_AL1342_Acyclic_Response;
	Request:cIFM_AL1342_Acyclic_Request;
	Response:cIFM_AL1342_Acyclic_Response;
	Acyclic_Request:BOOL;
	*)
	
END_STRUCT
END_TYPE

// Level_0/IO-Link/cIFM_AL1342
TYPE cIFM_AL1342 :
STRUCT
	Port_1_RX:ARRAY[0..15] OF WORD;
	Port_2_RX:ARRAY[0..15] OF WORD;
	Port_3_RX:ARRAY[0..15] OF WORD;
	Port_4_RX:ARRAY[0..15] OF WORD;
	Port_5_RX:ARRAY[0..15] OF WORD;
	Port_6_RX:ARRAY[0..15] OF WORD;
	Port_7_RX:ARRAY[0..15] OF WORD;
	Port_8_RX:ARRAY[0..15] OF WORD;
	
	Port_1_TX:ARRAY[0..15] OF WORD;
	Port_2_TX:ARRAY[0..15] OF WORD;
	Port_3_TX:ARRAY[0..15] OF WORD;
	Port_4_TX:ARRAY[0..15] OF WORD;
	Port_5_TX:ARRAY[0..15] OF WORD;
	Port_6_TX:ARRAY[0..15] OF WORD;
	Port_7_TX:ARRAY[0..15] OF WORD;
	Port_8_TX:ARRAY[0..15] OF WORD;
	
	Port_Request:ARRAY[1..8] OF 	cIFM_AL1342_Acyclic_Request;
	Port_Response:ARRAY[1..8] OF cIFM_AL1342_Acyclic_Response;
	Request:cIFM_AL1342_Acyclic_Request;
	Response:cIFM_AL1342_Acyclic_Response;
	Acyclic_Request:BOOL;
END_STRUCT
END_TYPE

// Level_0/SIO-MB04RTDS/cMB0_RTD
TYPE cMB0_RTD :
STRUCT
	//Temperature:ARRAY[0..3] OF Burkert.Burkert.cAIT;
	RX:cMB0_RTD_Raw_RX;
	TX:cMB0_RTD_Raw_TX;
END_STRUCT
END_TYPE

// Level_0/SIO-MB12CDR/cSIO_MB12CDR
TYPE cSIO_MB12CDR :
STRUCT
	Dout:ARRAY[0..4] OF BOOL;
	Din:ARRAY[0..7] OF BOOL;
	Frequency:ARRAY[0..3] OF REAL;
	Count:ARRAY[0..3] OF REAL;
	
	RX:cSIO_MB12CDR_RX;
	TX:cSIO_MB12CDR_TX;
END_STRUCT
END_TYPE

// VFD_CONTROL
TYPE VFD_CONTROL :
STRUCT
	MODE:uVFD_Mode;
	PLC_CMD	:REAL;
	PLC_Run:BOOL;
	MAN_CMD:REAL;
	Ready:BOOL;
	Actual:REAL;
	RunTime_Minutes:UDINT;
	Current_Alarm:Burkert.cAlarm_Config;
	Current_Status:Burkert.uSensor_Status;
	
END_STRUCT
END_TYPE

// VFD_GS2_DUT
TYPE VFD_GS2_DUT :
STRUCT
	CONTROL	:	VFD_Control;
	Status:	eVFD_Status;
	Output_Hz:REAL;
	Data:VFD_Status_Vacon_DUT;
END_STRUCT
END_TYPE

// VFD_WEG_DUT
TYPE VFD_WEG_DUT :
STRUCT
	CONTROL	:Burkert.VFD_Control;
	Status:eVFD_Status;
	Output_Hz:REAL;
	Data:VFD_Status_Weg_DUT;
END_STRUCT
END_TYPE

// cFilter
TYPE cFilter :
STRUCT
	Mode:uFilterMode;
	Status:eFilter_Status;
END_STRUCT
END_TYPE

// cFilter_Manager
TYPE cFilter_Manager :
STRUCT
	Mode:uFilter_Manager_Modes;
	Ststus:eFilter_Manager_Status;
	DP:Burkert.Burkert.cAIT;
	Filter_1:cFilter;
	Filter_2:cFilter;
	
END_STRUCT
END_TYPE

// Quick_Mix_Control
TYPE Quick_Mix_Control :
STRUCT
	Mode:uQuick_Mix_Modes;
	Status:eQuick_Mix_Status;
	Target_Volume:REAL:=250;
	Target_Temp:REAL:=85;
	Target_Rate:REAL:=75;
	ETA:UDINT;
	PLC_Run:BOOL;
	Active:BOOL;
	Ready:BOOL;
	CW_Valve:REAL;
	HW_Valve:REAL;
	
END_STRUCT
END_TYPE

// cPID_DUT
TYPE cPID_DUT EXTENDS PID_Control:
STRUCT
	
	
	KP:REAL:=1;
	TN:REAL:=0;
	TV:REAL:=0;
	CV_P:REAL;
	CV_I:REAL;
	CV_D:REAL;
	CV_FF:REAL;
	FF:REAL:=0;
	CV_Min:REAL:=0;
	CV_Max:REAL:=100;
	Live_Target:REAL;
	InHibit:BOOL;
END_STRUCT
END_TYPE

// cTempered_Line_Data
TYPE cTempered_Line_Data :
STRUCT
	Base_Flow:REAL;
	HW_Target_Flow:REAL;
	CW_Target_Flow:REAL;
	
	HW_CV:REAL;
	CW_CV:REAL;
	
	HW_DP:REAL;
	CW_DP:REAL;
	
	HW_FF:REAL;
	CW_FF:REAL;
	
	HW_KV:REAL;
	CW_KV:REAL;
	
	HW_Target_KV:REAL;
	CW_Target_KV:REAL;
	
	Target_Volume:REAL;
	Total_Volume:REAL;
	Flow_Rate:REAL;
	
	Target_Temperature:REAL;
	Temperature:REAL;
	//Temperature_Adjustment:REAL;
	
	
	CW_Flow_OK:BOOL;
	HW_Flow_OK:BOOL;
	Temperature_OK:BOOL;
	
	CW_Base_CV:REAL;
	HW_Base_CV:REAL;
	
	Max_Flow:REAL;
	Mode:eTempered_modes; 
	
	Status:uTempered_Status;
	StrStatus:STRING;
	
END_STRUCT
END_TYPE

// Level_3/Brewery/Brewery_Config_DUT
TYPE Brewery_Config_DUT :
STRUCT
	HLT:HLT_DUT;
	CLT:CLT_DUT;
	Grain_Room:GR_DUT;
	MM:MM_DUT;
	LTun:LT_DUT;
	KT:cKT;
	WP:cWP_DUT;
	Brew_Recipe:INT;
END_STRUCT
END_TYPE

// Burkert Library/Level_1/ACV_Modes
{attribute 'qualified_only'}
//{attribute 'strict'}
{attribute 'to_string'}
TYPE Burkert.eACV_Modes :
(
	Auto := 0,
	Closed,
	Open,
	Locate,
	xTune,
	Burkert_Open,//5
	Manual_Pos
	
	
);
END_TYPE

// Burkert Library/Level_1/AIT_Modes
{attribute 'qualified_only'}
//{attribute 'strict'}
{attribute 'to_string'}
TYPE Burkert.AIT_Modes :
(
	Active := 0,
	Forced,
	Alarms_Disabled,
	Alarm_Reset,
	OffLine
);
END_TYPE

// Burkert Library/Level_1/eBCV_Modes
{attribute 'qualified_only'}
//{attribute 'strict'}
{attribute 'to_string'}

TYPE eBCV_Modes :
(
	Auto:=0,
	Closed,
	Open,
	Identify,
	xTune,
	Burkert_Open //5
	
);
END_TYPE

// Burkert Library/Level_1/TT_Modes
{attribute 'qualified_only'}
//{attribute 'strict'}
TYPE Burkert.TT_Modes :
(
	Active := 0,
	Forced,
	Alarms_Disabled,
	Alarm_Reset,
	OffLine
);
END_TYPE

// Burkert Library/Level_1/eACV_Status
{attribute 'qualified_only'}
//{attribute 'strict'}
{attribute 'to_string'}

TYPE eACV_Status :
(
	A_Closed:=0,
	A_Open,
	M_Closed,
	M_Open,
	Opening, //
	Closing, //
	
	LOCKED_OUT,		//6
	Interlocked,	//
	OFFLINE,		//8
	
	Fault,		//
	Pos_Error,
	Error,// Namur 5	-,
		
		//
	Missing,
	Detected,
	P_Fault,
	Maintenance_Required,//Namur  2  
	Out_Of_Spec, //Namur 3	-
	Check_Function,//Namur 4	-
	Not_Used_Manual,
	A_Position,
	M_Position
				//
);
END_TYPE

// Burkert Library/Level_1/eBCV_Status
{attribute 'qualified_only'}
//{attribute 'strict'}
{attribute 'to_string'}

TYPE eBCV_Status :
(
	A_Closed := 0,
	A_Open,			//1
	M_Closed,
	M_Open,			//3
	Opening,
	Closing,//5
	LOCKED_OUT:=6,
	Interlocked,
	OFFLINE,
	
	Fault,		//9
	Both_Limits_Active,
	Error,// Namur 5
	
	Missing,	//12
	Detected,
	P_Fault,
	Maintenance_Required,//Namur  2  -15
	Out_Of_Spec, //Namur 3	-16
	Check_Function//Namur 4	-17


	
);
END_TYPE

// Burkert Library/Level_1/eSensor_Status
{attribute 'qualified_only'}
//{attribute 'strict'}
{attribute 'to_string'}
TYPE eSensor_Status :
(
	OK := 0,
	Low_Low_Alarm,
	Low_Warning,
	High_Warning,
	HiHi_Alarm,
	Offline, 
	FORCED,
	Alarms_Disabled,
	Under_Range,
	Over_Range,
	Missing,
	Detected,
	P_Fault,
	Fault
);
END_TYPE

// Burkert Librarry/Level_1/HMI_8050
TYPE HMI_8050 EXTENDS c8050 :
STRUCT
	strName:STRING;
	strMode:STRING;
	strStatus:STRING;
END_STRUCT
END_TYPE

// Burkert Librarry/Level_1/HMI_AIT
TYPE HMI_AIT EXTENDS Burkert.cAIT :
STRUCT
	strName:STRING;
	strMode:STRING;
	strStatus:STRING;
END_STRUCT
END_TYPE

// Burkert Librarry/Level_1/HMI_BCV
TYPE HMI_BCV EXTENDS Burkert.cBCV :
STRUCT
	strName:STRING;
	strMode:STRING;
	strStatus:STRING;
END_STRUCT
END_TYPE

// Burkert Librarry/Level_1/HMI_FIT
TYPE HMI_FIT EXTENDS Burkert.cFIT :
STRUCT
	strName:STRING;
	strMode:STRING;
	strStatus:STRING;
END_STRUCT
END_TYPE

// Burkert Librarry/Level_1/HMI_VFD_GS20_DUT
TYPE HMI_VFD_GS20_DUT EXTENDS cVFD_GS20_DUT :
STRUCT
	strName:STRING;
	strMode:STRING;
	strStatus:STRING;
END_STRUCT
END_TYPE

// Burkert Librarry/Level_1/HMI_VFD_Vacon_DUT
TYPE HMI_VFD_Vacon_DUT EXTENDS VFD_Vacon_DUT :
STRUCT
	strName:STRING;
	strMode:STRING;
	strStatus:STRING;
END_STRUCT
END_TYPE

// ceDip_ME44_DI
TYPE ceDip_ME44_DI  EXTENDS cME44_DI:
STRUCT
	RX:cME44_DI_RX;
	TX:cME44_DI_TX;
	strTCPstate:STRING[30];
	
	
END_STRUCT
END_TYPE

// cME44_DO
TYPE cME44_DO :
STRUCT
	Namur:BYTE;
	Dout:BYTE;
	RX_Namur:WORD;
	TX:cME44_DO_TX;
	
END_STRUCT
END_TYPE

// cME44_DO_TX
TYPE cME44_DO_TX :
STRUCT
		CH1Ch8:WORD;
		CH1Bin:WORD;
		CH2Bin:WORD;
		CH3Bin:WORD;
		CH4Bin:WORD;
		CH5Bin:WORD;
		CH6Bin:WORD;
		CH7Bin:WORD;
		CH8Bin:WORD;
		
		CH1Float:ARRAY[0..1] OF WORD;
		CH2Float:ARRAY[0..1] OF WORD;
		CH3Float:ARRAY[0..1] OF WORD;
		CH4Float:ARRAY[0..1] OF WORD;
		CH5Float:ARRAY[0..1] OF WORD;
		CH6Float:ARRAY[0..1] OF WORD;
		CH7Float:ARRAY[0..1] OF WORD;
		CH8Float:ARRAY[0..1] OF WORD;
		
		
		
END_STRUCT
END_TYPE

// In Burkert Device Library/LeveL_1/IO-Link/c8050
TYPE c8050 :
STRUCT
	CND:Burkert.Burkert.cAIT;
	Totalizer_1:REAL;
	Rate_1:Burkert.Burkert.cAIT;
	Temp:Burkert.Burkert.cAIT;
	PLC_Count_Reset:BOOL;
	HMI_Count_Reset:BOOL;
	strTCPstate:STRING[30];
END_STRUCT
END_TYPE

// cVFD_Eaton_DUT
TYPE cVFD_Eaton_DUT:// EXTENDS VFD_Control:
STRUCT
	CONTROL	:Burkert.VFD_Control;
	Status:uVFD_Status;
	Output_Hz:REAL;
	Output_Pct:REAL;
	Data:VFD_Status_Eaton_DUT;
	RX:ARRAY[0..10] OF WORD;	//Reg 42100
	TX:ARRAY[0..10] OF WORD;	//Reg 42000
	TCP_State:ModbusTCPComState;
	strTCPstate:STRING[30];
	
	
END_STRUCT
END_TYPE

// cNord_VFD
TYPE cNord_VFD :
STRUCT
	Mode:eVFD_Modes;
	eStatus:eVFD_Status;
	PLC_SP:REAL;
	PLC_Run:BOOL;
	MAN_SP:REAL;
	Status:cNord_Data_In;
	Control:cNord_Control_Word;
	SP_TX:INT;
	Ouput_PCT:REAL;
	//Network_Status:eCanInternalState;
	Node_ID:BYTE;
	
	
END_STRUCT
END_TYPE

// cVFD_STATUS_Vacon
TYPE cVFD_STATUS_Vacon :
STRUCT
Drive_STATUS:	VFD_Status_Word_DUT;
Status_code:INT;
//Output_Hz:REAL;
RPM:INT;
Motor_Current:REAL;
Motor_Torque:REAL;
Motor_Power:REAL;
Motor_Voltage:REAL;
DC_Link:REAL;
Fault_Code:INT;
Unit_Temperature:REAL;
//Network_Status:eChannelError;
END_STRUCT
END_TYPE

// cVFD_Vacon
TYPE cVFD_Vacon:// EXTENDS VFD_Control:
STRUCT
	CONTROL	:Burkert.VFD_Control;
	Status:uVFD_Status;
	Output_Hz:REAL;
	Output_Pct:REAL;
	Data:cVFD_Status_Vacon;
	TCP_State:ModbusTCPComState;
	strTCPstate:STRING[30];
	
	rx	:ARRAY[0..10] OF WORD;
	tx	:ARRAY[0..2] OF WORD;
END_STRUCT
END_TYPE

// cCellar_Vessel_Config_DUT
TYPE cCellar_Vessel_Config_DUT :
STRUCT
	Max_Capacity:REAL:=70000;	
	Current_Volume:REAL:=32000;
	Lower_Jacket_Top_PCT:REAL:=10;
	Middle_Jacket_Top_PCT:REAL:=55;
	Dead_Band:REAL:=0.25;
	//Error_Window:REAL:=1;
	//Alarm_Offset:Burkert.cAlarm_Offsets;
	Max_Cooling_Zones:INT:=3;
	PID_Index:				PID_Mapping;
	cSesnor_Index:			cSensor_Mapping;
	Alarm_Offset_index:		Alarm_Offset_Mapping;

	
	
	
	
	
	
END_STRUCT
END_TYPE

// cVessel_CIP
TYPE cVessel_CIP :
STRUCT
	Initial_Volume:REAL;
	Rate:REAL;
	Duration_S:UINT;	
END_STRUCT
END_TYPE

// cCLT_Assets
TYPE cCLT_Assets :
STRUCT
	Tank_LSHH: REFERENCE TO DI_DUT;
	Pump_Intake_LS	:REFERENCE TO DI_DUT;
	
	Tank_Level:		REFERENCE TO Burkert.cAIT;
	Temperature		:REFERENCE TO Burkert.cAIT;
	HTX_Discharge_TT	:REFERENCE TO Burkert.cAIT;
	Discharge_Pressure	:REFERENCE TO Burkert.cAIT;
	
	Recirc_FIT			:REFERENCE TO Burkert.cFIT;
	KT_FIT		:REFERENCE TO Burkert.cFIT;
	
	Recirc_ACV			:REFERENCE TO Burkert.cACV;
	Glycol_ACV			:REFERENCE TO Burkert.cACV;
	
	Fill_BCV			:REFERENCE TO Burkert.cBCV;
	
	PID_Recirc			:REFERENCE TO PID_DUT;
	PID_Temp			:REFERENCE TO PID_DUT;
	
	Pump:REFERENCE TO Burkert.VFD_Control;
	
	
	
	
END_STRUCT
END_TYPE

// CLT_DUT
TYPE CLT_DUT :
STRUCT
	Mode:uCLT_Mode;
	Task:uCLT_Task;
	Status:uCLT_Status;	
	AutoFill:CLT_AutoFill_Dut;
	recirc_Rate:REAL:=25;
	External_Demand:REAL;
	Profile:ARRAY[0..3] OF eCLT_Profile;
	//Assets:cCLT_Assets;
	
	StrMode:STRING;
	StrTask:STRING;
	StrStatus:STRING;
		
END_STRUCT
END_TYPE

// CLT_Profile
TYPE CLT_Profile :
STRUCT
	Level:Burkert.cAlarm_SetPoints;
	Temperature:Burkert.cAlarm_SetPoints;
	Enable_Hour:UINT;
	Enable_Minute:UINT;
	Enable_Days:WORD;
	Disable_Hour:UINT:=24;
	Disable_Minute:UINT:=00;
	
END_STRUCT
END_TYPE

// eCLT_Profile
TYPE eCLT_Profile :
STRUCT
	Level:Burkert.cAlarm_Config;
	Temperature:Burkert.cAlarm_Config;
	Enable_Time:UDINT;
	Enable_Days:WORD;
	
END_STRUCT
END_TYPE

// Heat_Profile_DUT
TYPE Heat_Profile_DUT :
STRUCT
	Upper_Temp:REAL:=65;
	Middle_Temp:REAL:=70;
	Lower_Temp:REAL:=75;
	Agitator_Speed:REAL:=20;
	Agitator_Speed_Rest:REAL:=20;
	Time_s:UINT:=600;
END_STRUCT
END_TYPE

// GR_DUT
TYPE GR_DUT :
STRUCT
	Mode:Burkert.uHOA_Mode;
	Task:uGR_Task;
	Status:uGR_Status;
	Fixed_Speed:REAL;
	Task_ETA:UINT;
	READY:BOOL;
	Hopper_Rate:REAL;
	
	StrMode:STRING;
	StrTask:STRING;
	StrStatus:STRING;
	
	
	//Assets:Grain_Room_Assets;
	
	
END_STRUCT
END_TYPE

// Grain_Room_Assets
TYPE Grain_Room_Assets :
STRUCT
	//Grain_Mill:Burkert.Contactor_DUT;
	//Conveyor_1:Burkert.Contactor_DUT;
	Conveyor_2:REFERENCE TO Burkert.VFD_Control;
	Hopper_Gate_Valve:REFERENCE TO Burkert.cBCV;
	Hydrator_Gate_Valve:REFERENCE TO Burkert.cBCV;
	
	Scale: REFERENCE TO Burkert.cAIT;
	
	
END_STRUCT
END_TYPE

// eHLT_Profile
TYPE eHLT_Profile :
STRUCT
	Level:Burkert.cAlarm_SetPoints;
	Temperature:Burkert.cAlarm_SetPoints;
	//Enable_Time:UDINT;
	Enable_Hour:UINT;
	Enable_Minute:UINT;
	Enable_Days:UINT;
	
	Disable_Hour:UINT:=24;
	Disable_Minute:UINT:=00;
	
END_STRUCT
END_TYPE

// eHLT_Setpoints
TYPE eHLT_Setpoints :
STRUCT
	Level:Burkert.cAlarm_SetPoints;
	Temperature:Burkert.cAlarm_SetPoints;
	//Enable_Time:UDINT;
	Enable_Hour:UINT;
	Enable_Minute:UINT;
	Enable_Days:UINT;
	
END_STRUCT
END_TYPE

// HLT_Assets
TYPE HLT_Assets :
STRUCT
	
	Strike_HW:REFERENCE TO Burkert.cACV;
	Strike_CW:REFERENCE TO Burkert.cACV;
	Sparge_HW:REFERENCE TO Burkert.cACV;
	Sparge_CW:REFERENCE TO Burkert.cACV;
	HTX_Outlet_ACV:REFERENCE TO Burkert.cACV;
	HTX_Steam:REFERENCE TO Burkert.cACV;
	
	
	Mix_Pump:REFERENCE TO Burkert.VFD_Control;
	Recirc_Pump:REFERENCE TO Burkert.VFD_Control;
	
	
	
	Strike_FIT:REFERENCE TO Burkert.cFIT;
	Sparge_FIT:REFERENCE TO Burkert.cFIT;
	HTX_FIT:REFERENCE TO Burkert.cFIT;
	//Service_Water_FIT:REFERENCE TO FIT_DUT;
	
	
	CW_Fill:REFERENCE TO Burkert.cBCV;
	Recirc_To_HTX:REFERENCE TO Burkert.cBCV;
	SprayBall:REFERENCE TO Burkert.cBCV;
	SW_Main_BCV: REFERENCE TO Burkert.cBCV;
	
	
	
	PID_HTX:REFERENCE TO cPID_DUT;
	PID_Recirc:REFERENCE TO cPID_DUT;
	//PID_Service_Water:REFERENCE TO PID_DUT;
	
	Temperature:REFERENCE TO Burkert.cAIT;
	Strike_TT:REFERENCE TO Burkert.cAIT;
	Sparge_TT:REFERENCE TO Burkert.cAIT;
	HTX_Outlet_TT:REFERENCE TO Burkert.cAIT;
	HTX_Inlet_TT:REFERENCE TO Burkert.cAIT;
	
	Mix_Pump_Pressure:REFERENCE TO Burkert.cAIT;
	Recirc_Pressure:REFERENCE TO Burkert.cAIT;
	Level:REFERENCE TO Burkert.cAIT;
	
	Pump_Intake_LSLL:REFERENCE TO DI_DUT;
	Tank_LSHH:REFERENCE TO DI_DUT;
	
	
	

	
END_STRUCT
END_TYPE

// ACV_Temp_Loop_UDFB
FUNCTION_BLOCK ACV_Temp_Loop_UDFB
VAR_IN_OUT
	ACV_LOOP: ACV_Temp_Loop_DUT;
	ACV:ACV_DUT;
	TT:AIT_DUT;

END_VAR

VAR_INPUT
	Heating: BOOL;
	LOCKOUT:BOOL:=FALSE;
	Permisive:BOOL:=TRUE;
	External_Fault:BOOL:=FALSE;
END_VAR
VAR

	FT_PID_0: BURKERT_OSCAT_BASIC.CTRL_PID;
	GEN_PULSE_0: BURKERT_OSCAT_BASIC.GEN_PULSE;
	In_Zone: BOOL;
	TON_0: TON;
	R_TRIG_0: R_trig;
	Timer_Status: INT;
	ABS_Error: REAL;
	R_TRIG_1: R_trig;
	RAMP_REAL_0: Util.RAMP_REAL;
	SR_0: SR;
	TON_1: TON;
	TOF_0: TOF;
	TON_2: TON;
	FT_PID_1:Util.PID_FIXCYCLE;
	Temp_Loop_PID:BOOL:=TRUE;
	R_trig_2:R_Trig;
	Loop_Disable:BOOL;
	TP_1:TP;
	
	FT_PIDW_1: BURKERT_OSCAT_BASIC.FT_PIDW;
END_VAR
VAR_OUTPUT

END_VAR
VAR // added by the converter: edge detectors and wires of the graphical bodies
    _w1, _w2, _w3, _w4, _w5, _w6, _w7, _w8, _w9, _w10, _w11, _w12, _w14 : ANY;
    _w13 : TIME;
END_VAR

// note: 7 stored wires end on pins the file does not list and are not shown
ACV_Loop.DeadBand := SEL(ACV_Loop.DeadBand = 0.0, ACV_Loop.DeadBand, 0.1);
ACV_Loop.Live_Target_EU := SEL(ACV_Loop.Mode=Temp_Loop_Modes.Step, ACV_Loop.Target_EU, SEL(HEATING, TT.EU-(ACV_Loop.DeadBand*1.5), TT.EU+(ACV_Loop.DeadBand*1.5)));
_w1 := (ACV_Loop.Mode = Temp_Loop_Modes.Crash) OR (ACV_Loop.Mode = Temp_Loop_Modes.Step);
_w2 := ABS(ACV_Loop.Target_Eu - TT.EU);
ABS_Error := _w2;
(* _w2 * ACV_Loop.kp < 50; result not used *)
TON_2(IN := False OR _w2 < (ACV_Loop.DeadBand*4), PT := T#5s); // TON
_w3 := _w1 AND TON_2.Q;
In_Zone := _w3;
R_TRIG_0(CLK := _w1 AND _w3); // R_trig
IF R_TRIG_0.Q THEN _w4 := Temp_Loop_Modes.Auto; END_IF
ACV_Loop.Mode := _w4;
_w5 := SEL(Heating, ACV_Loop.Live_Target_EU, ACV_Loop.Actual_EU);
ACV_Loop.Int_Out := FT_PIDW_1.YI;
_w6 := SEL(Heating, ACV_Loop.Actual_EU, ACV_Loop.Live_Target_EU);
TOF_0(IN := Permisive, PT := T#5s); // TOF
SR_0(SET1 := Loop_Disable, RESET := ACV_Loop.Mode=Temp_Loop_Modes.Idle); // SR
_w7 := (ACV_Loop.Mode=Temp_Loop_Modes.Auto_Paused) OR (ACV_Loop.Mode=Temp_Loop_Modes.Idle) OR NOT TOF_0.Q OR SR_0.Q1 OR (ACV_Loop.Status=Temp_Loop_Status.Timer_Expired) OR (TT.Status.eStatus=Burkert.eSensor_Status.Offline) OR (TT.Status.eStatus=Burkert.eSensor_Status.Fault) OR (acv.Status=Burkert.eACV_Status.OFFLINE);
_w8 := SEL(_w7, _w6, _w5) - _w5;
TP_1(IN := _w3, PT := T#5s); // TP
FT_PIDW_1(
    IN := _w8,
    KP := ACV_Loop.kp,
    TN := ACV_Loop.TN,
    TV := ACV_Loop.TV,
    LIM_L := 0,
    LIM_H := 100,
    RST := _w7 OR TP_1.Q); // BURKERT_OSCAT_BASIC.FT_PIDW
ACV_Loop.Limiter := FT_PIDW_1.LIM;
_w9 := SEL(ACV_Loop.Mode=Temp_Loop_Modes.Crash, FT_PIDW_1.Y, 100.0);
ACV_Loop.Diff_Out := FT_PIDW_1.diff.out;
_w10 := SEL(Loop_Disable, _w9, 0.0);
ACV.PLC_CMD := _w10;
ACV_Loop.Load_EU := _w10;
IF SR_0.Q1 THEN _w11 := Temp_Loop_Modes.Idle; END_IF
ACV_Loop.Mode := _w11;
TT.Burkert.cAlarm_Config.Hi_Hi_Alarm := SEL(NOT _w7, TT.Burkert.cAlarm_Config.Hi_Hi_Alarm, ACV_Loop.Live_Target_EU+(ACV_Loop.Window*2));
TT.Burkert.cAlarm_Config.Hi_Warn := SEL(NOT _w7, TT.Burkert.cAlarm_Config.Hi_Warn, ACV_Loop.Live_Target_EU+(ACV_Loop.Window));
TT.Burkert.cAlarm_Config.Low_warn := SEL(NOT _w7, TT.Burkert.cAlarm_Config.Low_warn, ACV_Loop.Live_Target_EU-(ACV_Loop.Window));
TT.Burkert.cAlarm_Config.Low_Low_Alarm := SEL(NOT _w7, TT.Burkert.cAlarm_Config.Low_Low_Alarm, ACV_Loop.Live_Target_EU-(ACV_Loop.Window*2));
ACV_Loop.Actual_EU := TT.EU;
ACV_Loop.Error_EU := SEL(ACV_Loop.Mode=Temp_Loop_Modes.Idle, TT.EU - ACV_Loop.Target_EU, 0.0);
_w12 := (ACV_Loop.Mode=Temp_Loop_Modes.Auto) AND (ACV_Loop.Timer_Target_M>0);
_w13 := UINT_TO_TIME(ACV_Loop.Timer_Target_M) * 60000;
TON_0(IN := _w12, PT := _w13); // TON
ACV_Loop.Timer_Remaining_s := TIME_TO_UINT((_w13 - TON_0.ET) / 1000);
_w14 := (TT.Status.eStatus=Burkert.eSensor_Status.Offline) OR (TT.Status.eStatus=Burkert.eSensor_Status.Fault) OR (acv.Status=Burkert.eACV_Status.OFFLINE);
Loop_Disable := External_Fault OR (TT.Status.eStatus=Burkert.eSensor_Status.FORCED) OR (ACV.Mode<>Burkert.eACV_Modes.Auto) OR _w14;
ACV_Loop.Status := SEL(ACV.Mode<>Burkert.eACV_Modes.Auto, SEL(TT.Status.eStatus=Burkert.eSensor_Status.FORCED, SEL(External_Fault, SEL(_w14, SEL(ACV_Loop.Mode=Temp_Loop_Modes.Auto_Paused, SEL(ACV_Loop.Mode=Temp_Loop_Modes.Idle, SEL(TT.Status.eStatus=Burkert.eSensor_Status.Low_Low_Alarm, SEL(TT.Status.eStatus=Burkert.eSensor_Status.Low_Warning, SEL(TT.Status.eStatus=Burkert.eSensor_Status.HiHi_Alarm, SEL(TT.Status.eStatus=Burkert.eSensor_Status.High_Warning, SEL(TON_0.Q, SEL(_w12, SEL(ACV_Loop.Mode=Temp_Loop_Modes.Auto, SEL(Permisive, Temp_Loop_Status.Pre_Start, Temp_Loop_Status.Ramping), Temp_Loop_Status.Auto), Temp_Loop_Status.Timed), Temp_Loop_Status.Timer_Expired), Temp_Loop_Status.HiHi_Warning), Temp_Loop_Status.HiHi_Alarm), Temp_Loop_Status.LoLo_Warning), Temp_Loop_Status.LoLo_Alarm), Temp_Loop_Status.Idle), Temp_Loop_Status.Paused), Temp_Loop_Status.Fault), Temp_Loop_Status.External_Fault), Temp_Loop_Status.Sensor_Forced), Temp_Loop_Status.Valve_Not_auto);
// TRUE: input not connected
// Temp_Loop_Status.Idle: input not connected

END_FUNCTION_BLOCK

// AODD_UDFB
FUNCTION_BLOCK AODD_UDFB
VAR
	Target_Rate: REAL;
	Base_On_Time: REAL;
	VPP: REAL;
	//TONOF_0: BURKERT_OSCAT_BASIC.TONOF;
	R_TRIG_0: R_trig;
	R_TRIG_1: R_Trig;
	Target_Volume: REAL;
	Shot_Count: INT;
	Calculated_On_Time:REAL;
	Base_Run_Time: REAL;
	TON_0: TON;
	//Pulse_0: BURKERT_OSCAT_BASIC.GEN_PULSE;
	TON_1: TON;
	Start_Volume: REAL;
	On_Off_Ratio:REAL;
	Required_Run_Time_S:REAL;
	Maximum_Shots:INT;
	Maximum_Shots_Run_Time_S:REAL;
	Maximum_Shots_Off_Time_S:REAL;
	Required_Run_Duration_S: REAL;
	Estimated_Run_Total_Run_Time_S:REAL;
	Volume_Per_Shot:REAL;
	Estimated_Total_Volume:REAL;
	//No_PWM: BOOL;
	CTD_0: CTD;
	R_TRIG_2: R_trig;
	F_TRIG_0: F_trig;
	TP_0: TP;
	TP_1: TP;
	TON_2: TON;
	TOF_0: TOF;
	FIRE: BOOL;
	Active: BOOL;
	TON_3: TON;
	F_TRIG_1: F_trig;
	F_TRIG_2: F_trig;
	START_Request: BOOL;
END_VAR
VAR_IN_OUT
	AODD:AODD_DUT;
END_VAR;
VAR_OUTPUT
	Q:BOOL;
END_VAR
VAR // added by the converter: edge detectors and wires of the graphical bodies
    _w1, _w2, _w4, _w5, _w13, _w14, _w16, _w18, _w19 : ANY;
    _w3 : BOOL;
    _w6, _w7, _w8, _w9, _w12, _w15 : INT;
    _w10, _w11 : REAL;
    _w17 : TIME;
END_VAR

_w1 := SEL(AODD.Mode=eAODD_Modes.Auto, SEL(NOT (AODD.Mode=eAODD_Modes.Auto), AODD.Base_Rate, AODD.HMI_Target_Rate), AODD.PLC_Target_Rate);
Target_Rate := _w1;
_w2 := _w1 / AODD.Base_Rate;
On_Off_Ratio := _w2;
_w3 := AODD.Min_On_Seconds / _w2 - AODD.Min_On_Seconds < AODD.Min_OFF_Seconds;
AODD.Duty_Cycle := _w2 * 100;
_w4 := SEL(AODD.Mode=eAODD_Modes.Auto, SEL(NOT (AODD.Mode=eAODD_Modes.Auto), 0, AODD.HMI_Target_Volume), AODD.PLC_Target_Volume);
Target_Volume := _w4;
Required_Run_Duration_S := _w4 / (Target_Rate/60);
_w5 := _w4 / (AODD.Base_Rate/60);
Required_Run_Time_S := _w5;
_w6 := _w5 / Maximum_Shots;
Maximum_Shots_Run_Time_S := _w6;
AODD.On_Time := _w6;
_w7 := (AODD.Base_Rate/60) * _w6;
Volume_Per_Shot := _w7;
Estimated_Total_Volume := Maximum_Shots * _w7;
_w8 := REAL_TO_INT(_w5 / AODD.Min_On_Seconds);
_w9 := SEL(_w3 OR _w8 = 0, _w8, 1);
Maximum_Shots := _w9;
_w10 := Required_Run_Duration_S / _w9 - _w6;
_w11 := SEL(_w10 < 0, _w10, 0);
Maximum_Shots_Off_Time_S := _w11;
AODD.Off_Time := _w11;
Estimated_Run_Total_Run_Time_S := Maximum_Shots * (_w6 + _w11);
Set_Status();
_w12 := SEL(start_Request, 0.0, (Maximum_Shots - AODD.Shots_Remaining) * (aodd.On_Time*(Aodd.Base_Rate/60)));
_w13 := (AODD.Mode=eAODD_Modes.Manual) OR (AODD.Mode=eAODD_Modes.Auto) AND aodd.PLC_Run;
START_Request := _w13;
TON_3(IN := _w13, PT := T#2s); // TON
F_TRIG_2(CLK := _w13); // F_trig
R_TRIG_0(CLK := _w13); // R_trig
_w14 := F_TRIG_2.Q OR R_TRIG_0.Q;
_w15 := SEL(_w14, _w12, 0.0);
F_TRIG_1(CLK := Fire); // F_trig
R_TRIG_2(CLK := _w13); // R_trig
CTD_0(CD := F_TRIG_1.Q, LOAD := R_TRIG_2.Q, PV := Maximum_Shots); // CTD
AODD.Shots_Remaining := CTD_0.CV;
_w16 := TON_3.Q AND NOT CTD_0.Q;
Active := _w16;
_w17 := REAL_TO_TIME(SEL(Maximum_Shots=1, Maximum_Shots_Off_Time_S, 5) * 1000);
_w18 := _w16 AND NOT TOF_0.Q;
TON_2(IN := _w18, PT := REAL_TO_TIME(Maximum_Shots_Run_Time_S * 1000)); // TON
_w19 := _w16 AND _w18 AND NOT TON_2.Q;
FIRE := _w19;
Start_Volume := SEL(_w14, SEL(_w19, AODD.Volume_Delivered, Start_Volume), _w15);
TON_1(IN := _w19, PT := T#30m); // TON
AODD.Volume_Delivered := SEL(_w19, _w15, Start_Volume + (TIME_TO_REAL(TON_1.ET) / 1000) * (AODD.Base_Rate/60));
TOF_0(IN := TON_2.Q, PT := _w17); // TOF
Q := (AODD.Mode=eAODD_Modes.Prime) OR _w19;

END_FUNCTION_BLOCK

// Basic_Temp_LOOP
FUNCTION_BLOCK Basic_Temp_LOOP
VAR	
	RS_0: RS;
END_VAR
VAR_IN_OUT
	Loop:BCV_Temp_Loop_DUT;
END_VAR
VAR_INPUT
END_VAR
VAR // added by the converter: edge detectors and wires of the graphical bodies
    _w1 : ANY;
END_VAR

_w1 := Loop.Target_EU + Loop.Window;
RS_0(SET := loop.Actual_EU > Loop.DeadBand + _w1, RESET1 := loop.Actual_EU < _w1 - Loop.DeadBand); // RS
Loop.Output := RS_0.Q1;

END_FUNCTION_BLOCK

// BCV_Temp_Loop_UDFB
FUNCTION_BLOCK BCV_Temp_Loop_UDFB
VAR_IN_OUT
	BCV_LOOP: BCV_Temp_Loop_DUT;
	BCV:BCV_DUT;
	TT:AIT_DUT;

END_VAR

VAR_INPUT
	Heating: BOOL;
	LOCKOUT:BOOL:=FALSE;
	Permisive:BOOL:=TRUE;
	External_Fault:BOOL:=FALSE;
	//Temp_Loop_PID:WORD:=2;
	//BCV_ID:INT;
	//TT_ID:INT;
END_VAR
VAR

